(* CODESYS project AnimalCT.project
   Title: AnimalCT
   CompiledLibraryCompatibilityVersion: LeadSysStudio V3.5 SP15 Patch 4

Project tree, tasks and I/O mapping:
  Device : MC508, Leadshine Technology Co., Ltd., order no. 508101, version 3.5.15.40
      settings: RetainMode = 0; RetainStartAddr = 20480; RetainEndAddr = 524288; RetainSize = 524288
    application Application
      libraries: Standard, * (System); CAA SerialCom, 3.5.15.0 (CAA Technical Workgroup); Serial Communication, 3.5.7.0 (3S - Smart Software Solutions GmbH); LS_SysLib, 1.0.0.9 (Leadshine Technology Co.Ltd); CANopenLib, 1.0.0.5 (Leadshine Technology Co.Ltd); CAA Net Base Services, 3.5.15.0 (CAA Technical Workgroup); Network, 3.5.7.0 (3S - Smart Software Solutions GmbH); CANbus, 3.5.7.0 (3S - Smart Software Solutions GmbH); VisuDialogs, * (System); LS_OmronUtils, 1.0.0.2 (Leadshine Technology Co.Ltd); CANopenLib, 1.0.0.5 (Leadshine Technology Co.Ltd); SysMem23, 3.5.13.0 (System); SysFile, 3.5.15.0 (System); SysTypes2 Interfaces, 3.5.4.0 (System)
      task EtherCAT_Master_Leadshine_A (cyclic, interval 4 ms, priority 0) calls EtherCAT_Master_Leadshine_A.EtherCAT_Task, Axis_QJ, Axis_XZ
      task X_Ray (cyclic, interval t#4ms, priority 1) calls DT_Xray
      task MainTask (cyclic, interval 4 ms, priority 1) calls PLC_PRG
      DTU/
        data type E_State
        Axis/
          data type AxisState
          data type AxisCmd
          data type AxisParameter
        TCP/
          data type PLC_SEND
          data type PLC_RECV
          data type Real_TO_Byte_Convert
        data type E_LampCmd
      GVL/
        global variables GVL_Retain
        global variables GVL_SCAN
        global variables GVL_State
      BasicFBs/
        function block Blink [ST]
        function block MoveFilter [ST]
        function block ASCII_Chart_N [ST]
        function block RC [ST]
        function block Curve_Cs [ST]
        function block ASCII_Chart_P [ST]
        function block MeanValue [ST]
        function block Cut [ST]
        function block String2Byte [ST]
      RecordLog/
        program RecordLog [ST]: ACT_RecordState, ACT_RecordError, ACT_RecordCmd, ACT_XrayState, ACT_SysFileOpen, ACT_SysFileRename, ACT_SysFileRead, ACT_SysFileDelete, ACT_SysFileSetPos, ACT_SysFileWrite, ACT_SysFileClose, ACT_SysFileEOF, ACT_SysFileGetPos, ACT_SysFileCopy, ACT_RecordSwitch
      program DT_Xray [SFC]: _Error_active, T_Exp, _Serial_active, T_DR, T_Flu, _aOpenSeria_active, _Exposure1_active, _Wait_active, _Exposure2_entry, _Exposure2_active, _a_Init_active, _QueryState_entry, _Debug_active, _Exposure1_entry, _QueryState_active, _DefaultPara_entry, _DefaultPara_active, _a_DrExposure_active_1, _a_DrExposure_entry_1, _a_DrPara_active_1, _a_DrPara_entry_1, _a_FluoroPara_active_1, _a_FluoroPara_entry_1, _a_FluoroExPosure_active_1, _a_FluoroExPosure_entry_1, _a_ExposurePara_active_1, _a_ExposurePara_entry_1, _a_Exposure_active_1, _a_Exposure_entry_1, _Error_entry, _QueryState_exit, _a_FluoroExPosure_exit
      Refer/
        program Trigger_HaoboPannel [ST]
        program WriteLog [ST]: ACT_SysFileRead, ACT_SysFileDelete, ACT_SysFileClose, ACT_SysFileRename, ACT_SysFileGetPos, ACT_SysFileCopy, ACT_SysFileSetPos, ACT_SysFileEOF, ACT_SysFileWrite, ACT_SysFileOpen
        program XRAY_RS485 [ST]: AXray
      trace Trace (task MainTask): WorkStation_TCP.PLC_RECV1.m_nSocketType, Entity_IO.bXaryOne, Entity_IO.bXaryTwo, Entity_IO.bXaryFlu, Entity_IO.bXrayExp, Entity_IO.bTriggerOut, DT_Xray.RadExp_Step, PLC_PRG.Step_Scout, PLC_PRG.Step_CBCT, WorkStation_TCP.PLC_SEND1.m_nMHuValue, PLC_PRG.Step_StaticDR, WorkStation_TCP.PLC_RECV1.m_nLastMsg, Entity_IO.bXrayOneInput, WorkStation_TCP.PLC_SEND1.m_nMoveState, PLC_PRG.iActNumPulse, PLC_PRG.Step_Air, Entity_IO.bDoorLock, PLC_PRG.Step_QuickCT, GVL_State.iPLC_State
      global variables PersistentVars
      Init/
        program InitMotor [ST]
      visualisation Motor
      program PLC_PRG [SFC]: _a_SelfCheck_active, _a_StandardCT_active, _a_ShutDown_entry_1, T_JUMP_IDLE, _a_StaticDR_exit, _a_Emergercy_active_1, _a_StaticCT_active, _a_Idle_exit, T_StaticDR, T_DynamicsDR, _a_Idle_entry, _a_StaticCT_entry, T_CT, _a_SelfCheck_exit, _a_Error_entry, T_QuickCT, _a_Error_active, _a_HighDefinCT_active, _a_Homing_active, _a_Emergercy_entry_1, _a_QuickCT_exit, T_StandardCT, _a_SelfCheck_entry, AirHigh_entry, T_HighDefinCT, _a_DynamicsDR_exit, _a_Init_active_1, _a_ShutDown_active_1, _a_DynamicsDR_active, _a_Wait_active, _a_Idle_active, _a_Error_exit, _a_HighDefinCT_exit, _a_Homing_entry, _a_Debug_entry, _a_Init_active, _a_Logic_active, _a_Wait_exit, _a_StaticDR_active, _a_QuickCT_entry, _a_StandardCT_entry, _a_StaticCT_exit, _a_SystemInfo_active, _a_HighDefinCT_entry, _a_Debug_active, T_DR, _a_DynamicsDR_entry, _a_Homing_exit, _a_QuickCT_active, _a_MovePos_active, _a_StandardCT_exit, T_StaticCT, _a_StaticDR_entry, AirHigh_active, T_AirCal, T_AirCal_Quick, _AirCalQuick_active, _AirCalQuick_entry, _AirCalHign_exit, _AirCalQuick_exit, _a_Debug_exit, _a_Emergercy_exit, _ModeWait_active
      Logic/
        program WorkMode [ST]
      Motor/
        program Axis_XZ [ST]
        program Axis_QJ [ST]
        program Motor_SJ [ST]
      aSpecailBasic/
        function String2ASCII [ST]
        function block X_RayExpPara [ST]
        function block RecvStringS [ST]
        function block SendStringS [ST]
        function block X_RayFluPara [ST]
        function block String_TO_ASCII [ST]
      visualisation Entity_IO
      Communication/
        program CTBOX_RS232 [ST]
        program Calibration [ST]
        program WorkStation_TCP [ST]: APLC_RECV, APLC_SENG
      IOs/
        program Entity_IO [ST]
    Resource Usage
    Device Diagnose
    Network Configuration
      LocalBus Config
    EtherCAT_Master_Leadshine_A : EtherCAT Master SoftMotion, 3S - Smart Software Solutions GmbH, version 3.5.15.30
        settings: SlaveAutoRestart = True; NetworkName = 'ecat'; SelectNetworkByName = TRUE
      L8EC : L8EC(COE), Leadshine Technology Co.,Ltd., order no. L8EC, version Revision=16#00000001
          settings: StationAlias = 0; DC sync0 cycletime = 4000; DC sync1 cycletime = 4000; Number of SDO = 6; Homing method.Index = 16#6098; Homing method.Subindex = 16#00; Homing method.Value = 13; Homing method.Size = 8; Homing method.AbortIfError = FALSE; Homing method.JumpToLine = FALSE; Homing method.Line = 0; Homing method.CompleteAccess = False; Homing velocity (fast).Index = 16#6099; Homing velocity (fast).Subindex = 16#01; Homing velocity (fast).Value = 82451; Homing velocity (fast).Size = 32; Homing velocity (fast).AbortIfError = FALSE; Homing velocity (fast).JumpToLine = FALSE; Homing velocity (fast).Line = 0; Homing velocity (fast).CompleteAccess = False; Homing velocity (slow).Index = 16#6099; Homing velocity (slow).Subindex = 16#02; Homing velocity (slow).Value = 20612; Homing velocity (slow).Size = 32; Homing velocity (slow).AbortIfError = FALSE; Homing velocity (slow).JumpToLine = FALSE; Homing velocity (slow).Line = 0; Homing velocity (slow).CompleteAccess = False; Homing acceleration.Index = 16#609A; Homing acceleration.Subindex = 16#00; Homing acceleration.Value = 2576613; Homing acceleration.Size = 32; Homing acceleration.AbortIfError = FALSE; Homing acceleration.JumpToLine = FALSE; Homing acceleration.Line = 0; Homing acceleration.CompleteAccess = False; Homing offset.Index = 16#607C; Homing offset.Subindex = 16#00; Homing offset.Value = 0; Homing offset.Size = 32;
            Homing offset.AbortIfError = FALSE; Homing offset.JumpToLine = FALSE; Homing offset.Line = 0; Homing offset.CompleteAccess = False
          input  bRotateMotorMin1 : BOOL  // Digital inputs.Bit0
          input  bRotateMotorMax1 : BOOL  // Digital inputs.Bit1
          unmapped channels: Control word, Profile target position, Touch Probe Function, Servo error code, Last error code, Status word, Modes of operation display, Actual motor position, Touch Probe Status, Touch probe pos1 pos value, Digital inputs
        Axis : Axis, 3S - Smart Software Solutions GmbH, order no. 0, version 4.6.1.0
            settings: wDriveID = 0; dwRatioTechUnitsDenom = 432871; iRatioTechUnitsNum = 42; 一圈脉冲数 = 229167; 工作台一圈的位移 = 360; 电子齿轮比分子 = 340; 电子齿轮比分母 = 21; 回零速度 = 8.000; 回零爬行速度 = 2; 回零加速度 = 250.000; 回零偏移 = 0; 回零速度SDO = 82451; 回零爬行速度SDO = 20612; 回零偏移SDO = 0; ScalingIncs = 229167; ScalingMotorTurns2 = 340; ScalingGearOutput1 = 21; AdrOffset_8010 = 52; BitOffset_8010 = 0; BitLength_8010 = 16; Address_8010 = '%QW26'; Type_8010 = 'UINT'; AddressPointer_8010 = ADR(%QW26); AdrOffset_8020 = 56; BitOffset_8020 = 0; BitLength_8020 = 32; Address_8020 = '%QD14'; Type_8020 = 'DINT'; AddressPointer_8020 = ADR(%QD14); AdrOffset_8030 = 4294967295; BitOffset_8030 = 0; BitLength_8030 = 0; Address_8030 = ''; Type_8030 = ''; AddressPointer_8030 = 0; AdrOffset_8040 = 4294967295; BitOffset_8040 = 0; BitLength_8040 = 0; Address_8040 = ''; Type_8040 = '';
              AddressPointer_8040 = 0; AdrOffset_8050 = 4294967295; BitOffset_8050 = 0; BitLength_8050 = 0; Address_8050 = ''; Type_8050 = ''; AddressPointer_8050 = 0; AdrOffset_8060 = 60; BitOffset_8060 = 0; BitLength_8060 = 16; Address_8060 = '%QW30'; Type_8060 = 'UINT'; AddressPointer_8060 = ADR(%QW30); AdrOffset_8070 = 4294967295; BitOffset_8070 = 0; BitLength_8070 = 0; Address_8070 = ''; Type_8070 = ''; AddressPointer_8070 = 0; AdrOffset_8080 = 4294967295; BitOffset_8080 = 0; BitLength_8080 = 0; Address_8080 = ''; Type_8080 = ''; AddressPointer_8080 = 0; AdrOffset_8090 = 4294967295; BitOffset_8090 = 0; BitLength_8090 = 0; Address_8090 = ''; Type_8090 = ''; AddressPointer_8090 = 0; AdrOffset_8510 = 88; BitOffset_8510 = 0; BitLength_8510 = 16; Address_8510 = '%IW44'; Type_8510 = 'UINT'; AddressPointer_8510 = ADR(%IW44); AdrOffset_8520 = 92; BitOffset_8520 = 0; BitLength_8520 = 32;
              Address_8520 = '%ID23'; Type_8520 = 'DINT'; AddressPointer_8520 = ADR(%ID23); AdrOffset_8530 = 4294967295; BitOffset_8530 = 0; BitLength_8530 = 0; Address_8530 = ''; Type_8530 = ''; AddressPointer_8530 = 0; AdrOffset_8540 = 4294967295; BitOffset_8540 = 0; BitLength_8540 = 0; Address_8540 = ''; Type_8540 = ''; AddressPointer_8540 = 0; AdrOffset_8550 = 90; BitOffset_8550 = 0; BitLength_8550 = 8; Address_8550 = '%IB90'; Type_8550 = 'SINT'; AddressPointer_8550 = ADR(%IB90); AdrOffset_8560 = 104; BitOffset_8560 = 0; BitLength_8560 = 32; Address_8560 = '%ID26'; Type_8560 = 'UDINT'; AddressPointer_8560 = ADR(%ID26); AdrOffset_8570 = 96; BitOffset_8570 = 0; BitLength_8570 = 16; Address_8570 = '%IW48'; Type_8570 = 'UINT'; AddressPointer_8570 = ADR(%IW48); AdrOffset_8580 = 100; BitOffset_8580 = 0; BitLength_8580 = 32; Address_8580 = '%ID25'; Type_8580 = 'DINT'; AddressPointer_8580 = ADR(%ID25); AdrOffset_8590 = 4294967295;
              BitOffset_8590 = 0; BitLength_8590 = 0; Address_8590 = ''; Type_8590 = ''; AddressPointer_8590 = 0; AdrOffset_8600 = 4294967295; BitOffset_8600 = 0; BitLength_8600 = 0; Address_8600 = ''; Type_8600 = ''; AddressPointer_8600 = 0; AdrOffset_8600 = 4294967295; BitOffset_8600 = 0; BitLength_8600 = 0; Address_8610 = ''; Type_8610 = ''; AddressPointer_8610 = 0; AdrOffset_8620 = 4294967295; BitOffset_8620 = 0; BitLength_8620 = 0; Address_8620 = ''; Type_8620 = ''; AddressPointer_8620 = 0; 回零加速度SDO = 2576613
      L8EC_1 : L8EC(COE), Leadshine Technology Co.,Ltd., order no. L8EC, version Revision=16#00000001
          settings: StationAlias = 0; DC sync0 cycletime = 4000; DC sync1 cycletime = 4000; Number of SDO = 6; Homing method.Index = 16#6098; Homing method.Subindex = 16#00; Homing method.Value = 1; Homing method.Size = 8; Homing method.AbortIfError = FALSE; Homing method.JumpToLine = FALSE; Homing method.Line = 0; Homing method.CompleteAccess = False; Homing velocity (fast).Index = 16#6099; Homing velocity (fast).Subindex = 16#01; Homing velocity (fast).Value = 60000; Homing velocity (fast).Size = 32; Homing velocity (fast).AbortIfError = FALSE; Homing velocity (fast).JumpToLine = FALSE; Homing velocity (fast).Line = 0; Homing velocity (fast).CompleteAccess = False; Homing velocity (slow).Index = 16#6099; Homing velocity (slow).Subindex = 16#02; Homing velocity (slow).Value = 12000; Homing velocity (slow).Size = 32; Homing velocity (slow).AbortIfError = FALSE; Homing velocity (slow).JumpToLine = FALSE; Homing velocity (slow).Line = 0; Homing velocity (slow).CompleteAccess = False; Homing acceleration.Index = 16#609A; Homing acceleration.Subindex = 16#00; Homing acceleration.Value = 100000; Homing acceleration.Size = 32; Homing acceleration.AbortIfError = FALSE; Homing acceleration.JumpToLine = FALSE; Homing acceleration.Line = 0; Homing acceleration.CompleteAccess = False
          input  bForeMotorMin1 : BOOL  // Digital inputs.Bit0
          input  bForeMotorMax1 : BOOL  // Digital inputs.Bit1
          unmapped channels: Control word, Profile target position, Touch Probe Function, Servo error code, Last error code, Status word, Modes of operation display, Actual motor position, Touch Probe Status, Touch probe pos1 pos value, Digital inputs
        Axis_1 : Axis, 3S - Smart Software Solutions GmbH, order no. 0, version 4.6.1.0
            settings: dwRatioTechUnitsDenom = 2000; 一圈脉冲数 = 20000; 工作台一圈的位移 = 10; 电子齿轮比分子 = 1; 电子齿轮比分母 = 1; 回零速度 = 30.000; 回零爬行速度 = 6.000; 回零加速度 = 50; 回零偏移 = 0; 回零速度SDO = 60000; 回零爬行速度SDO = 12000; ScalingIncs = 20000; AdrOffset_8010 = 64; BitOffset_8010 = 0; BitLength_8010 = 16; Address_8010 = '%QW32'; Type_8010 = 'UINT'; AddressPointer_8010 = ADR(%QW32); AdrOffset_8020 = 68; BitOffset_8020 = 0; BitLength_8020 = 32; Address_8020 = '%QD17'; Type_8020 = 'DINT'; AddressPointer_8020 = ADR(%QD17); AdrOffset_8030 = 4294967295; BitOffset_8030 = 0; BitLength_8030 = 0; Address_8030 = ''; Type_8030 = ''; AddressPointer_8030 = 0; AdrOffset_8040 = 4294967295; BitOffset_8040 = 0; BitLength_8040 = 0; Address_8040 = ''; Type_8040 = ''; AddressPointer_8040 = 0; AdrOffset_8050 = 4294967295; BitOffset_8050 = 0; BitLength_8050 = 0; Address_8050 = '';
              Type_8050 = ''; AddressPointer_8050 = 0; AdrOffset_8060 = 72; BitOffset_8060 = 0; BitLength_8060 = 16; Address_8060 = '%QW36'; Type_8060 = 'UINT'; AddressPointer_8060 = ADR(%QW36); AdrOffset_8070 = 4294967295; BitOffset_8070 = 0; BitLength_8070 = 0; Address_8070 = ''; Type_8070 = ''; AddressPointer_8070 = 0; AdrOffset_8080 = 4294967295; BitOffset_8080 = 0; BitLength_8080 = 0; Address_8080 = ''; Type_8080 = ''; AddressPointer_8080 = 0; AdrOffset_8090 = 4294967295; BitOffset_8090 = 0; BitLength_8090 = 0; Address_8090 = ''; Type_8090 = ''; AddressPointer_8090 = 0; AdrOffset_8510 = 112; BitOffset_8510 = 0; BitLength_8510 = 16; Address_8510 = '%IW56'; Type_8510 = 'UINT'; AddressPointer_8510 = ADR(%IW56); AdrOffset_8520 = 116; BitOffset_8520 = 0; BitLength_8520 = 32; Address_8520 = '%ID29'; Type_8520 = 'DINT'; AddressPointer_8520 = ADR(%ID29); AdrOffset_8530 = 4294967295; BitOffset_8530 = 0;
              BitLength_8530 = 0; Address_8530 = ''; Type_8530 = ''; AddressPointer_8530 = 0; AdrOffset_8540 = 4294967295; BitOffset_8540 = 0; BitLength_8540 = 0; Address_8540 = ''; Type_8540 = ''; AddressPointer_8540 = 0; AdrOffset_8550 = 114; BitOffset_8550 = 0; BitLength_8550 = 8; Address_8550 = '%IB114'; Type_8550 = 'SINT'; AddressPointer_8550 = ADR(%IB114); AdrOffset_8560 = 128; BitOffset_8560 = 0; BitLength_8560 = 32; Address_8560 = '%ID32'; Type_8560 = 'UDINT'; AddressPointer_8560 = ADR(%ID32); AdrOffset_8570 = 120; BitOffset_8570 = 0; BitLength_8570 = 16; Address_8570 = '%IW60'; Type_8570 = 'UINT'; AddressPointer_8570 = ADR(%IW60); AdrOffset_8580 = 124; BitOffset_8580 = 0; BitLength_8580 = 32; Address_8580 = '%ID31'; Type_8580 = 'DINT'; AddressPointer_8580 = ADR(%ID31); AdrOffset_8590 = 4294967295; BitOffset_8590 = 0; BitLength_8590 = 0; Address_8590 = ''; Type_8590 = ''; AddressPointer_8590 = 0;
              AdrOffset_8600 = 4294967295; BitOffset_8600 = 0; BitLength_8600 = 0; Address_8600 = ''; Type_8600 = ''; AddressPointer_8600 = 0; AdrOffset_8600 = 4294967295; BitOffset_8600 = 0; BitLength_8600 = 0; Address_8610 = ''; Type_8610 = ''; AddressPointer_8610 = 0; AdrOffset_8620 = 4294967295; BitOffset_8620 = 0; BitLength_8620 = 0; Address_8620 = ''; Type_8620 = ''; AddressPointer_8620 = 0; 回零加速度SDO = 100000
    LocalBus_Master_Module : LocalBus Master, Leadshine Technology Co., Ltd., version 3.5.15.40
      PM_3200 : PM_3200, Leadshine Technology Co., Ltd., version 3.5.15.40
          settings: 位置号 = 0
          unmapped channels: ErrorCode, INPUT_0, INPUT_1
      PM0016R : PM0016R, Leadshine Technology Co., Ltd., version 3.5.15.40
          settings: 位置号 = 1
          unmapped channels: ErrorCode, OUTPUT_0
      PM_A0400_IV : PM_A0400_IV, Leadshine Technology Co., Ltd., version 3.5.15.40
          settings: 位置号 = 2; AD0 config.Data_Buffer = 5; AD1 config.Data_Buffer = 5; AD2 config.Data_Buffer = 5; AD3 config.Data_Buffer = 5
          unmapped channels: ErrorCode, ADValue, AnalogDiagnose
    Free_Protocol_RS232_COM : Free Protocol RS232 COM, Leadshine Technology Co., Ltd., version 3.5.15.40
        settings: Vendor.Baudrate = 19200; Vendor.Parity = 2; max send data count = 20; max receive data count = 20; com interval = 25
        unmapped channels: receive control, receive data size, send control, send data size, send data buffer, error status, error id, actual receive data size, actual send data size, receive data
    High_Speed_IO_Module : High Speed IO, Leadshine Technology Co., Ltd., version 3.5.15.40
        settings: HS_IO_Mode_0.High In IO Mode 4 = 196611; HS_IO_Mode_0.High In IO Mode 5 = 196611; Counter_Mask = 48; Ioin_Mask = 1792; HS counter 6.Counter_SetWorkMode = 2; InputFilter Para.Time_In8 = 10; InputFilter Para.Time_In9 = 10; InputFilter Para.Time_In10 = 10
        unmapped channels: Genral_IO_IN, Genral_IO_Out
    SoftMotion General Axis Pool
    Free_Protocol_RS485_COM : Free Protocol RS485 COM, Leadshine Technology Co., Ltd., version 3.5.15.40
        settings: Vendor.Baudrate = 19200; Vendor.Parity = 2; max send data count = 10; max receive data count = 10; com interval = 50
        unmapped channels: receive control, receive data size, send control, send data size, send data buffer, error status, error id, actual receive data size, actual send data size, receive data
  text list GlobalTextList
*)

// Device/Application/DTU/TCP/PLC_SEND
TYPE PLC_SEND:
	STRUCT
		m_nSocketType		:UDINT;	//心跳指令，默认为3，留待判断连接状态。
		m_nCurrentAngle		:REAL;	//为设备当前的旋转角度，单位为角度制下的单位，为度。数精度为1度；
		m_nBedHeight		:REAL;	//为床高，单位为毫米，数据范围为0 - 2000mm；
		m_nBedMovePos		:REAL;	//为床移动距离，以床与探测板的垂直面交线为起点，单位为毫米，数据范围为0 - 3000mm；
		m_nExpStates		:UDINT;	//为曝光状态，枚举值，0:idle（空闲） 1:prep（训机） 2: ready（训机结束，准备完成，可以出束） 3: XrayOn（出射线） 4:XrayOff（关射线） 5 error；
		m_nExpCount			:UDINT;	//为曝光的次数，对应曝光的图像张数；
		m_nFocus			:UDINT;	//按键提示，物理意义更改为按键提示
		m_nMHuValue			:REAL;	//热容量，单位MHu ，实际热容量*100得到，实际热容量为小数；
		m_nDirectionState	:UDINT;	//当前旋转状态，默认值-1， 0为正转，1为反转，停止为-1
		m_nMoveState		:UDINT;	//起始、终止状态， 默认值-1， 0为当前扫描方案（与常规意义不同，注意区别）处于准备好状态，可以准备扫描；1为当前扫描方案结束，运动过程中值为-1
		m_nError			:UDINT;	//错误码使用，由王（风杰）工具体阐述内容
		m_fSpeed			:REAL;	//为设备的旋转速度，单位为度/秒，精度0.01度/秒；
		m_fKv				:UDINT;	//管电压，单位为kv（千伏），精度1；
		m_fMA				:REAL;	//管电流，单位为mA（毫安），精度0.1；
		m_fMs				:REAL;	//曝光时间，单位为ms（毫秒），精度0.01；
		m_nSamplingRate		:UDINT;	//采样率，有3个选项：2400帧/圈；1200帧/圈；600帧/圈
		m_nScanProType		:UDINT;	//执行扫描方案的类型，0为自动扫描，1为手动扫描，2为无设置意义的值，默认值为2
		PLC_State			:UDINT;	//PLC状态
		XRAY_State			:UDINT;	//X射线源状态
		AxisErrorID			:UDINT;	//电机错误标志位，含2个伺服电机
		
		m_nFocusX			:UDINT;	//焦点大小，0为大焦点 1为小焦点， 焦点具体对应的值由plc设置；
		reserve1,reserve2,reserve3,reserve4,reserve5,reserve6,reserve7,reserve8,reserve9:UDINT;
	END_STRUCT
END_TYPE

// Device/Application/DTU/E_State
{attribute 'qualified_only'}
{attribute 'strict'}
TYPE E_State :
(
	初始化		:=10,
	自检		:=20,
	回零		:=30,
	待机 		:=40,
	静态DR		:=110,
	动态DR		:=120,
	标准CT		:=210,
	静态CT 		:=220,
	高清CT		:=230,
	快速CT		:=240,
	错误状态	:=310,
	调试状态 	:=320,
	急停状态	:=330,
	关机状态	:=340
);
END_TYPE

// Device/Application/DTU/TCP/PLC_RECV
TYPE PLC_RECV :
	STRUCT
		m_nSocketType		:UDINT;//0为连接判断信息使用，1为发送设备的有具体意义是参数信息。
      	m_nExpId 			:UDINT;//扫描方式 0为不扫描， 1为静态DR扫描 2为动态DR扫描，3为标准CT，4为静态CT，5为高清CT，6为快速CT
       	m_nAngleStart 		:REAL;//为曝光起始位置，在2D和多次曝光情况下，机架旋转到m_nAngleStart位置后再开始曝光，机架不动；CBCT状态下，机架旋转到m_nAngleStart位置后开始曝光，机架运动至m_nAngleEnd位置；最小值为0。
      	m_nAngleEnd  		:REAL;//为曝光的终止位置，在2D和多次曝光情况下不使用；在CBCT状态下，机架的运动终止位置；最小值为0，最大值为360。
      	m_nRotateBegin  	:REAL;//为旋转的起始位置（考虑加速过程）
      	m_nRotateEnd  		:REAL;//为旋转的终止位置（考虑减速过程）
      	m_nKv  				:UDINT;//设置的管电压值，单位为kv，正整数；
      	m_nMA  				:REAL;//设置的管电流值，单位为mA，正整数；
      	m_nMS 				:REAL;//设置一次曝光的时间，单位为ms（毫秒）；设置一次曝光的时间，单位为us（微秒）；精度为1
       	m_nFocus 			:UDINT;//焦点大小设置，枚举值，0为大焦点， 1小焦点；
      	m_nAcquireFrame 	:UDINT;//总帧数，正整数；
      	m_nFramePerCirCle	:UDINT;//每圈获得的帧数，正整数，帧/圈；
      	m_nMoveToward  		:UDINT;//扫描方向，0为不移动，1为进床方向，2为出床方向；
     	m_nServenLamp  		:UDINT;//七灯是否点亮
      	m_nMoveStep  		:REAL;//步进长度，轴扫时使用，单位为mm（毫米）；
     	m_nPitchValue   	:REAL;//螺距长度，螺旋扫时使用，单位为mm（毫米）；
      	m_nCircleCount  	:UDINT;//旋转总圈数，由起始角度和终止角度计算获得，正整数。
      	m_nControlState 	:UDINT;//控制状态 0为正常 1为中止扫描， 2为退出扫描，默认为0
       	m_fScanTop 			:REAL;//扫描上界，以动物趴卧头朝里的方向为基准，从脚至头方向为正方向。单位为毫米，精度为0.01；
       	m_fScanBottom 		:REAL;//扫描下界，以动物趴卧头朝里的方向为基准，从脚至头方向为正方向。单位为毫米，精度为0.01；
		m_fSecondPerCicle	:REAL;//一圈多少秒
      	m_nSamplingRate  	:UDINT;//采样率，有3个选项：2400帧/圈；1200帧/圈；600帧/圈
       	m_nPrepareState 	:UDINT;//是否亮灯1为亮5灯，0 为不亮5灯
        m_nScanMoveType		:UDINT;//扫描模式 0为手动扫描，1为自动扫描，2为子床位扫描
       	m_nCircleIndex 		:UDINT;//当前第几圈
       	m_nPLCMaCoeff 		:REAL;//灯丝电压值
      	m_nLastMsg  		:UDINT;//CBCT扫描最后一次标志位
       	m_nDelayTime 		:UDINT;//预留
        yuliu_2				:UDINT;//预留
       	yuliu_3 			:UDINT;//预留一共30个数据
	END_STRUCT
END_TYPE

// Device/Application/DTU/E_LampCmd
{attribute 'qualified_only'}
{attribute 'strict'}
TYPE E_LampCmd :
(
	常亮	:=66,
	慢闪	:=22,
	快闪	:=33,
	关闭 	:=55
);
END_TYPE

// Device/Application/DTU/TCP/Real_TO_Byte_Convert
	(*共用体，2个16位WORD和转换为REAL类型*)
	TYPE Real_TO_Byte_Convert :
	UNION
		rData:REAL;					//32字节
		wByte:ARRAY[0..3] OF BYTE;  //8位字节
	END_UNION
	END_TYPE

// Device/Application/DTU/Axis/AxisState
TYPE AxisState :
STRUCT
	bNetState	:BOOL;//网络状态
	bStandStill	:BOOL;//静止状态
	bPowering	:BOOL;//使能状态
	bHoming		:BOOL;//回零状态
	bErrStop	:BOOL;//停止错误
	bStopState	:BOOL;//停止状态
	bAxisErr	:BOOL;//轴故障
	bPowerOff	:BOOL;//轴使能中
	bContinuousMotion:BOOL;//连续运动状态
	bDisCreteMition:BOOL;//离散运动状态
	bSynchronizedMotion:BOOL;//同步运动中
	
	bAxisGoAbsDone	:BOOL;//绝对定位完成10ms后自动复位
	bAxisGoRelDone	:BOOL;//相对定位完成10ms后自动复位
	bResetDone		:BOOL;//复位完成
	
	rActPosition	:LREAL; 	//实际位置
	rActVelocity	:LREAL; 	//实际速度
	rActTorque		:LREAL;	//实际力矩
	rAcc			:REAL;	//加速度数值
	ErrorID			:UDINT;//故障代码
	
END_STRUCT
END_TYPE


(*
	dActPosition	:DINT; 	//实际位置
	dActVelocity	:DINT; 	//实际速度
	dActTorque		:DINT;	//实际力矩
	dAcc			:DINT;	//加速度数值
*)

// Device/Application/DTU/Axis/AxisCmd
TYPE AxisCmd :
STRUCT
	bPower	: BOOL;	//上电使能
	bHome	: BOOL;	//上升沿触发，10ms后自动复位，请勿一致强制ON
	bJogP	: BOOL;	//正向点动
 	bJogN	: BOOL;	//反向点动
	bAbs	: BOOL;	//上升沿触发，10ms后自动复位，请勿一致强制ON
	bRel	: BOOL;	//上升沿触发，10ms后自动复位，请勿一致强制ON
	bVel	: BOOL;  //速度模式 	
	bStop	: BOOL;	//停止
	bReset	: BOOL;//上升沿触发，10ms后自动复位，请勿一致强制ON
	bSetPos	:BOOL;//设置轴当前位置,home
	bSetPosH:BOOL;//setPos
	AxisPara: AxisParameter;
	bSetHomePara:BOOL;//设置回零参数
END_STRUCT
END_TYPE

// Device/Application/DTU/Axis/AxisParameter
TYPE AxisParameter :
STRUCT
	AxisNodeID			: USINT;	
	rZeroOffset			: REAL;//回原点偏移
	rAbsPosition		: REAL;//AxisGoAbs位置
	rAbsVelocity		: REAL;	//AxisGoAbs速度
	rRelVelocity		: REAL;//AxisGoRel速度
	rRelPosition		: REAL;//AxisGoRel位置
	rVelVelocity		: REAL;//AxisVGo速度
	rAccDec				: REAL;//加减速
	rJogVelocity		: REAL;//点动加减速度默认为点动速度10倍
	rSetPosition		: REAL;//设置轴当前位置变量
	
	iHomeMode		:USINT;
	rHomeHighSpeed	:REAL;
	rHomeLowSpeed	:REAL;
	rHomeAcc		:REAL;
END_STRUCT
END_TYPE


(*	
STRUCT
	AxisNodeID			: USINT;	
	dZeroOffset			: UDINT;//回原点偏移
	dAbsPosition		: DINT;//AxisGoAbs位置
	dAbsVelocity		: UDINT;	//AxisGoAbs速度
	dRelVelocity		: UDINT;//AxisGoRel速度
	dRelPosition		: DINT;//AxisGoRel位置
	dVelVelocity		: DINT;//AxisVGo速度
	dAccDec				: UDINT;//加减速
	dJogVelocity		: DINT;//点动加减速度默认为点动速度10倍
	dSetPosition		: UDINT;//设置轴当前位置变量
	
	iHomeMode		:USINT;
	dHomeHighSpeed	:UDINT;
	dHomeLowSpeed	:UDINT;
	dHomeAcc		:UDINT;
END_STRUCT
*)

// Device/Application/GVL/GVL_Retain
{attribute 'qualified_only'}

VAR_GLOBAL PERSISTENT RETAIN
	rBedRecordHeight:REAL;//断电保存
	rBedRecordLength:REAL;//断电保存
	
	rXZ_Zero:REAL;
	rSJ_Zero:INT;
	
	
	rXZ_Position:REAL;
	rQJ_Position:REAL;
END_VAR

// Device/Application/GVL/GVL_SCAN
{attribute 'qualified_only'}
VAR_GLOBAL
		bJumpScan:BOOL;
END_VAR

// Device/Application/PersistentVars
{attribute 'qualified_only'}	//掉电保持数据

// Device/Application/GVL/GVL_State
{attribute 'qualified_only'}
VAR_GLOBAL
		iPLC_State:UDINT;
		
		iXray_State:UDINT; 
	
END_VAR

// Device/Application/Motor/Axis_QJ
PROGRAM Axis_QJ
VAR
	
	fbMC_Power			:	MC_Power;
	fbMC_Jog			: 	MC_Jog;
	fbMC_Stop			: 	MC_STOP;	
	fbMC_Home			:	MC_HOME;
	fbMC_Reset			:	MC_Reset;
	fbMC_MoveAbsolute	: 	MC_MoveAbsolute;
	fbMC_MoveRelative	: 	MC_MoveRelative;
	fbMC_ReadStatus		:	MC_ReadStatus;
	fbMC_ReadActualPosition:MC_ReadActualPosition;
	fbMC_ReadActualVelocity	:MC_ReadActualVelocity;
	fbMC_ReadActualTorque:MC_ReadActualTorque;
	fbMC_MoveVelocity:MC_MoveVelocity;
	fbMC_SetPostiong:		MC_SetPosition;
	count				:	BYTE;
	VelDirection:INT:=1;
END_VAR

VAR_INPUT
	QJ_AxisCmd			:AxisCmd;
END_VAR

VAR_OUTPUT	
	QJ_AxisState 		:AxisState;
END_VAR

(*--------------README----------*)
(*旋转电机运动子程序*)

(*1.心跳*)
	count:=count+1;
				
(*2.判断电机轴状态*)
	fbMC_ReadStatus(Axis:= AXIS_1, Enable:= TRUE , //周期刷新
					valid=> , 
					Busy=> , 
					Error=> QJ_AxisState.bAxisErr,   	//轴错误
					ErrorID=> QJ_AxisState.ErrorID,  	//错误ID
					ErrorStop=>QJ_AxisState.bErrStop , 	//轴停止
					Disabled=> QJ_AxisState.bPowerOff, 	//轴未使能
					stopping=> QJ_AxisState.bStopState, //轴紧急停止
					Homing=>	QJ_AxisState.bHoming , 		//回零中
					Standstill=> QJ_AxisState.bStandStill, //使能中
					DiscreteMotion=> QJ_AxisState.bDisCreteMition, 		//离散运动中
					ContinuousMotion=>QJ_AxisState.bContinuousMotion );	//持续运动中
					
		
(*3 读取轴当前位置、速度*)
(*3.1 获取当前位置*)
	fbMC_ReadActualPosition(
								Axis:= AXIS_1, 
								Enable:= TRUE, 
								Valid=> , 
								Busy=> , 
								Error=> , 
								ErrorID=> , 
								Position=> QJ_AxisState.rActPosition);
(*3.2 获取当前速度*)	
	fbMC_ReadActualVelocity(
								Axis:= AXIS_1 ,
								Enable:= TRUE, 
								Valid=> , 
								Busy=> , 
								Error=> , 
								ErrorID=> , 
								Velocity=> QJ_AxisState.rActVelocity);
(*3.3 获取当前力矩*)								
	fbMC_ReadActualTorque(
								Axis:= AXIS_1 ,
								Enable:= TRUE, 
								Valid=> , 
								Busy=> , 
								Error=> , 
								ErrorID=> , 
								Torque=> );
	QJ_AxisState.rActTorque:=fbMC_ReadActualTorque.Torque*1270/1000;						
(*4.使能*)
	fbMC_Power(
				Axis:= AXIS_1 ,
				Enable:= TRUE, 
				bRegulatorOn:= QJ_AxisCmd.bPower,  
				bDriveStart:= QJ_AxisCmd.bPower,  
				Status=>  QJ_AxisState.bPowering, 
				bRegulatorRealState=> , 
				bDriveStartRealState=> , 
				Busy=> , 
				Error=> , 
				ErrorID=> );
	
(*5.回零*)
	fbMC_Home(
				Axis:= AXIS_1, 
				Execute:= QJ_AxisCmd.bHome, 
				Position:= 0,				//回零模式1，默认写零
				Done=> , 
				Busy=> , 
				CommandAborted=> , 
				Error=> , 
				ErrorID=> );
				
(*6.设置当前位置*)			
	fbMC_SetPostiong(
						Axis:= AXIS_1, 
						Execute:= QJ_AxisCmd.bSetPos, 
						Position:= GVL_Retain.rQJ_Position, //设置当前位置
						Mode:= FALSE, 
						Done=> , 
						Busy=> , 
						Error=> , 
						ErrorID=> );
	
(*6.速度模式*)
(*	IF QJ_AxisCmd.AxisPara.rVelVelocity>0 THEN
			VelDirection:=1;
		ELSE
			VelDirection:=-1;
		END_IF
	fbMC_MoveVelocity(
					Axis:=AXIS_1 , 
					Execute:=  QJ_AxisCmd.bVel, 
					Velocity:=ABS(QJ_AxisCmd.AxisPara.rVelVelocity), 
					Acceleration:= QJ_AxisCmd.AxisPara.rAccDec, 
					Deceleration:= QJ_AxisCmd.AxisPara.rAccDec, 
					Jerk:= QJ_AxisCmd.AxisPara.rAccDec*10, 
					Direction:= VelDirection, 
					BufferMode:= 0, 
					InVelocity=> , 
					Busy=> , 
					Active=> , 
					CommandAborted=> , 
					Error=> , 
					ErrorID=> );
*)
(*7.轴绝对运动*)
	fbMC_MoveAbsolute(
						Axis:= AXIS_1, 
						Execute:= QJ_AxisCmd.bAbs AND (NOT QJ_AxisState.bStopState), 
						Position:= QJ_AxisCmd.AxisPara.rAbsPosition, 
						Velocity:= QJ_AxisCmd.AxisPara.rAbsVelocity, 
						Acceleration:= QJ_AxisCmd.AxisPara.rAccDec, 
						Deceleration:= QJ_AxisCmd.AxisPara.rAccDec, 
						Jerk:= QJ_AxisCmd.AxisPara.rAccDec*10, 
						Direction:= 1, 
						BufferMode:= 0, 
						Done=> , 
						Busy=> , 
						Active=> , 
						CommandAborted=> , 
						Error=> , 
						ErrorID=> );
	
						
(*8.轴相对运动*)
	fbMC_MoveRelative(
						Axis:= AXIS_1, 
						Execute:= QJ_AxisCmd.bRel, 
						Distance:= QJ_AxisCmd.AxisPara.rRelPosition, 
						Velocity:=  QJ_AxisCmd.AxisPara.rRelVelocity, 
						Acceleration:=  QJ_AxisCmd.AxisPara.rAccDec, 
						Deceleration:=  QJ_AxisCmd.AxisPara.rAccDec, 
						Jerk:= QJ_AxisCmd.AxisPara.rAccDec*10, 
						BufferMode:= 0, //中断
						Done=> , 
						Busy=> , 
						Active=> , 
						CommandAborted=> , 
						Error=> , 
						ErrorID=> );
						
(*9.轴点动*)
	fbMC_Jog(
				Axis:= AXIS_1 ,
				JogForward:=  QJ_AxisCmd.bJogP AND (NOT QJ_AxisCmd.bJogN),
				JogBackward:= QJ_AxisCmd.bJogN AND (NOT QJ_AxisCmd.bJogP),
				Velocity:= QJ_AxisCmd.AxisPara.rJogVelocity,
				Acceleration:= QJ_AxisCmd.AxisPara.rAccDec, 
				Deceleration:= QJ_AxisCmd.AxisPara.rAccDec, 
				Jerk:= QJ_AxisCmd.AxisPara.rAccDec*10, 
				Busy=> , 
				CommandAborted=> , 
				Error=> , 
				ErrorId=> );

(*10.轴停止*)
	fbMC_Stop(
				Axis:= AXIS_1 ,
				Execute:=  QJ_AxisCmd.bStop, 
				Deceleration:= QJ_AxisCmd.AxisPara.rAccDec, 
				Jerk:= QJ_AxisCmd.AxisPara.rAccDec*10, 
				Done=> , 
				Busy=> , 
				Error=> , 
				ErrorID=> );

	IF fbMC_Stop.Done OR fbMC_Stop.Error THEN
		QJ_AxisCmd.bStop:=FALSE;
	END_IF

(*11.轴复位*)
	fbMC_Reset(
				Axis:= AXIS_1, 
				Execute:= QJ_AxisCmd.bReset, 
				Done=> QJ_AxisState.bResetDone, 
				Busy=> , 
				Error=> , 
				ErrorID=> );

END_PROGRAM

// Device/Application/Motor/Axis_XZ
PROGRAM Axis_XZ
VAR
	
	fbMC_Power			:	MC_Power;
	fbMC_Jog			: 	MC_Jog;
	fbMC_Stop			: 	MC_STOP;	
	fbMC_Home			:	MC_HOME;
	fbMC_Reset			:	MC_Reset;
	fbMC_MoveAbsolute	: 	MC_MoveAbsolute;
	fbMC_MoveRelative	: 	MC_MoveRelative;
	fbMC_ReadStatus		:	MC_ReadStatus;
	fbMC_ReadActualPosition:MC_ReadActualPosition;
	fbMC_ReadActualVelocity	:MC_ReadActualVelocity;
	fbMC_ReadActualTorque	:MC_ReadActualTorque;
	fbMC_MoveVelocity:		MC_MoveVelocity;
	fbMC_SetPostiong:		MC_SetPosition;
	VelDirection:INT:=1;
	count				:	BYTE;
	rLoadTorque:REAL;//负载力矩
END_VAR

VAR_INPUT
	XZ_AxisCmd			:AxisCmd;
END_VAR

VAR_OUTPUT	
	XZ_AxisState 		:AxisState;
END_VAR

(*--------------README----------*)
(*旋转电机运动子程序*)

(*1.心跳*)
	count:=count+1;
				
(*2.判断电机轴状态*)
	fbMC_ReadStatus(Axis:= Axis, Enable:= TRUE , //周期刷新
					valid=> , 
					Busy=> , 
					Error=> XZ_AxisState.bAxisErr,   	//轴错误
					ErrorID=> XZ_AxisState.ErrorID,  	//错误ID
					ErrorStop=>XZ_AxisState.bErrStop , 	//轴停止
					Disabled=> XZ_AxisState.bPowerOff, 	//轴未使能
					stopping=> XZ_AxisState.bStopState, //轴紧急停止
					Homing=>XZ_AxisState.bHoming , 		//回零中
					Standstill=> XZ_AxisState.bStandStill, //使能中
					DiscreteMotion=> XZ_AxisState.bDisCreteMition, 		//离散运动中
					ContinuousMotion=>XZ_AxisState.bContinuousMotion );	//持续运动中
					
		
(*3 读取轴当前位置、速度*)
(*3.1 获取当前位置*)
	fbMC_ReadActualPosition(
								Axis:= AXIS, 
								Enable:= TRUE, 
								Valid=> , 
								Busy=> , 
								Error=> , 
								ErrorID=> , 
								Position=> XZ_AxisState.rActPosition);
(*3.2 获取当前速度*)	
	fbMC_ReadActualVelocity(
								Axis:= AXIS, 
								Enable:= TRUE, 
								Valid=> , 
								Busy=> , 
								Error=> , 
								ErrorID=> , 
								Velocity=> XZ_AxisState.rActVelocity);
(*3.3 获取当前力矩*)								
	fbMC_ReadActualTorque(
								Axis:= AXIS, 
								Enable:= TRUE, 
								Valid=> , 
								Busy=> , 
								Error=> , 
								ErrorID=> , 
								Torque=> );
	XZ_AxisState.rActTorque:=fbMC_ReadActualTorque.Torque*2390/1000;//换算成mNM,额定力矩2.39NM ,反馈0.1%
	
	rLoadTorque:=LREAL_TO_REAL(XZ_AxisState.rActTorque)*371/1000;
								
(*4.使能*)
	fbMC_Power(
				Axis:= AXIS, 
				Enable:= TRUE, 
				bRegulatorOn:=  XZ_AxisCmd.bPower, 
				bDriveStart:=  XZ_AxisCmd.bPower, 
				Status=> XZ_AxisState.bPowering, 
				bRegulatorRealState=> , 
				bDriveStartRealState=> , 
				Busy=> , 
				Error=> , 
				ErrorID=> );
	
(*5.回零*)
	fbMC_Home(
				Axis:= AXIS, 
				Execute:= XZ_AxisCmd.bHome, 
				Position:= GVL_Retain.rXZ_Zero, 
				Done=> , 
				Busy=> , 
				CommandAborted=> , 
				Error=> , 
				ErrorID=> );
	
(*6.设置当前位置*)
	fbMC_SetPostiong(
						Axis:= AXIS, 
						Execute:= XZ_AxisCmd.bSetPos, 
						Position:= GVL_Retain.rXZ_Position, 
						Mode:= FALSE, 
						Done=> , 
						Busy=> , 
						Error=> , 
						ErrorID=> );
(*6.速度模式*)
(*	IF XZ_AxisCmd.AxisPara.rVelVelocity>0 THEN
		VelDirection:=1;
	ELSE
		VelDirection:=-1;
	END_IF
	fbMC_MoveVelocity(
				Axis:=AXIS , 
				Execute:=  XZ_AxisCmd.bVel, 
				Velocity:= ABS(XZ_AxisCmd.AxisPara.rVelVelocity), 
				Acceleration:= XZ_AxisCmd.AxisPara.rAccDec, 
				Deceleration:= XZ_AxisCmd.AxisPara.rAccDec, 
				Jerk:= XZ_AxisCmd.AxisPara.rAccDec*10, 
				Direction:= VelDirection, 
				BufferMode:= 0, 
				InVelocity=> , 
				Busy=> , 
				Active=> , 
				CommandAborted=> , 
				Error=> , 
				ErrorID=> );
*)
(*7.轴绝对运动*)
	fbMC_MoveAbsolute(
						Axis:= Axis, 
						Execute:= XZ_AxisCmd.bAbs AND (NOT XZ_AxisState.bStopState), 
						Position:= XZ_AxisCmd.AxisPara.rAbsPosition, 
						Velocity:= XZ_AxisCmd.AxisPara.rAbsVelocity, 
						Acceleration:= XZ_AxisCmd.AxisPara.rAccDec, 
						Deceleration:= XZ_AxisCmd.AxisPara.rAccDec, 
						Jerk:= XZ_AxisCmd.AxisPara.rAccDec*10, 
						Direction:= 1, 
						BufferMode:= 0, 
						Done=> , 
						Busy=> , 
						Active=> , 
						CommandAborted=> , 
						Error=> , 
						ErrorID=> );
	
						
(*8.轴相对运动*)
	fbMC_MoveRelative(
						Axis:= Axis, 
						Execute:= XZ_AxisCmd.bRel, 
						Distance:= XZ_AxisCmd.AxisPara.rRelPosition, 
						Velocity:=  XZ_AxisCmd.AxisPara.rRelVelocity, 
						Acceleration:=  XZ_AxisCmd.AxisPara.rAccDec, 
						Deceleration:=  XZ_AxisCmd.AxisPara.rAccDec, 
						Jerk:= XZ_AxisCmd.AxisPara.rAccDec*10, 
						BufferMode:= 0, //中断
						Done=> , 
						Busy=> , 
						Active=> , 
						CommandAborted=> , 
						Error=> , 
						ErrorID=> );
						
(*9.轴点动*)
	fbMC_Jog(
				Axis:= AXIS, 
				JogForward:=  XZ_AxisCmd.bJogP AND (NOT XZ_AxisCmd.bJogN),
				JogBackward:= XZ_AxisCmd.bJogN AND (NOT XZ_AxisCmd.bJogP),
				Velocity:= XZ_AxisCmd.AxisPara.rJogVelocity,
				Acceleration:= XZ_AxisCmd.AxisPara.rAccDec, 
				Deceleration:= XZ_AxisCmd.AxisPara.rAccDec, 
				Jerk:= XZ_AxisCmd.AxisPara.rAccDec*10, 
				Busy=> , 
				CommandAborted=> , 
				Error=> , 
				ErrorId=> );

(*10.轴停止*)
	fbMC_Stop(
				Axis:= AXIS, 
				Execute:=  XZ_AxisCmd.bStop, 
				Deceleration:= XZ_AxisCmd.AxisPara.rAccDec, 
				Jerk:= XZ_AxisCmd.AxisPara.rAccDec*10, 
				Done=> , 
				Busy=> , 
				Error=> , 
				ErrorID=> );

	IF fbMC_Stop.Done OR fbMC_Stop.Error THEN
		XZ_AxisCmd.bStop:=FALSE;
	END_IF

(*11.轴复位*)
	fbMC_Reset(
				Axis:= Axis, 
				Execute:= XZ_AxisCmd.bReset, 
				Done=> XZ_AxisState.bResetDone, 
				Busy=> , 
				Error=> , 
				ErrorID=> );

END_PROGRAM

// Device/Application/DT_Xray
PROGRAM DT_Xray
VAR
	Open_0: COM.Open;
	Write_0: COM.Write;
	Read_0: COM.Read;
	Close_0: COM.Close;
	hComHandle:CAA.HANDLE;
	aParamsB19200 : ARRAY [1..7] OF COM.PARAMETER := [
    (udiParameterId := COM.CAA_Parameter_Constants.udiPort,udiValue := 3), 					//指令端口2,3,4,5分别对应硬件接口com2、com0、com1、com3
    (udiParameterId := COM.CAA_Parameter_Constants.udiBaudrate,udiValue := 19200),			//波特率，设置为19200
    (udiParameterId := COM.CAA_Parameter_Constants.udiParity,udiValue := COM.PARITY.NONE),	//校验，设置为无校验
    (udiParameterId := COM.CAA_Parameter_Constants.udiStopBits,udiValue := COM.STOPBIT.ONESTOPBIT),//停止位，1位
    (udiParameterId := COM.CAA_Parameter_Constants.udiTimeout,udiValue := 500),				//超时时间，设置成500ms
    (udiParameterId := COM.CAA_Parameter_Constants.udiByteSize,udiValue := 8),				//数据位
    (udiParameterId := COM.CAA_Parameter_Constants.udiBinary, udiValue := 1)				//二进制参数，启用二进制模式
];		
	bSend: BOOL;//发送触发
	TON1,TON2,TON3:Standard.TON;//延迟打开串口，读取状态周期，初始态故障复位
	byReadData:ARRAY [0..255] OF BYTE; //读取串口数据
	xClose_Exe: BOOL; //关闭串口操作
	
	ReadString:RecvStringS;//读取射线源反馈，并转化为字符串型数据
	
	Lookup_Step:INT:=0;//查询状态的轮询
	BLINK1,BLINK1_ST,BLINK1_1S:Blink;
	
	SendStringS1:SendStringS;//单命令字符串发送
	
	ASCII_Chart_N2:ARRAY[0..30] OF ASCII_Chart_N;//解析查询态下的ASCII
	ASCII_Chart_N_Alarm:ARRAY[0..5] OF ASCII_Chart_N;//解析报警状态下的故障码
	ASCII_Chart_N_Alarm1,ASCII_Chart_N_Alarm2,ASCII_Chart_N_Alarm3:ASCII_Chart_N;
	(*透视写参变量*)
	FluParaSet:X_RayFluPara;//透视模式下的大指令写入
	String_TO_ASCII1:String_TO_ASCII;	//大命令字符串转化为ASCII码，给计算和校验用的
	ArrASCII:ARRAY[1..255] OF BYTE;		//ASCII放到数组里	
	CheckSum,CheckSum1,CheckSum2:UINT;//和校验处理
	CheckSum3,CheckSum4,CheckSum5:UINT;//和校验处理
	CheckSumString:STRING;//计算后的和校验后1个byte转化为字符串类型
	j,k:INT;//计算和校验用的//HE热量
	sSendStringFlu:STRING;//发送透视模式下的大命令
	TON_HangOver:TON;
	
	(*曝光写参变量*)
	ExpParaSet:X_RayExpPara;//透视模式下的大指令写入
	R_TRIG1,R_TRIG2,R_TRIG3,R_TRIG4,R_TRIG5,R1,R2,R3,R_Error:R_TRIG;
	bXrayError,bXrayError1: BOOL;//射线源出错标志位
	iDR_Staiton:UINT; //DR模式下的BU0选择，选择不同的站模式
	TON11,TON12,TON13,TON14:TON;//曝光跳出
	TOF11:TOF;
	bJumpRadExp:BOOL;
	
	Step_Error:INT;//错误回复步骤
	TOF_DR1:Standard.TOF;//延迟断电继电器控制
	
	
	bResetXray1:BOOL;
	bResetXray2:BOOL;
	sResetError,sResetError1,sResetError2,sResetError3,sResetError4:STRING;
END_VAR

VAR_OUTPUT
	iXray_State:INT;//射线源状态，改用全局变量
	Init_Step,Default_Step,Query_Step,RadExp_Step,RadFlu_Step,ExpPara_Step,FluPara_Setp,DR_Step,DR_Para:INT;//子状态
	Feedback_Kv:UDINT;
	Feedback_mA:REAL;
	Feedback_ms:REAL;
	Feedback_nFocus:UDINT;
	Feedback_nMHuValue:REAL;
	Feedback_AccTime:REAL;
	iAlarmNum:UINT;		//射线源部分的报警位
END_VAR

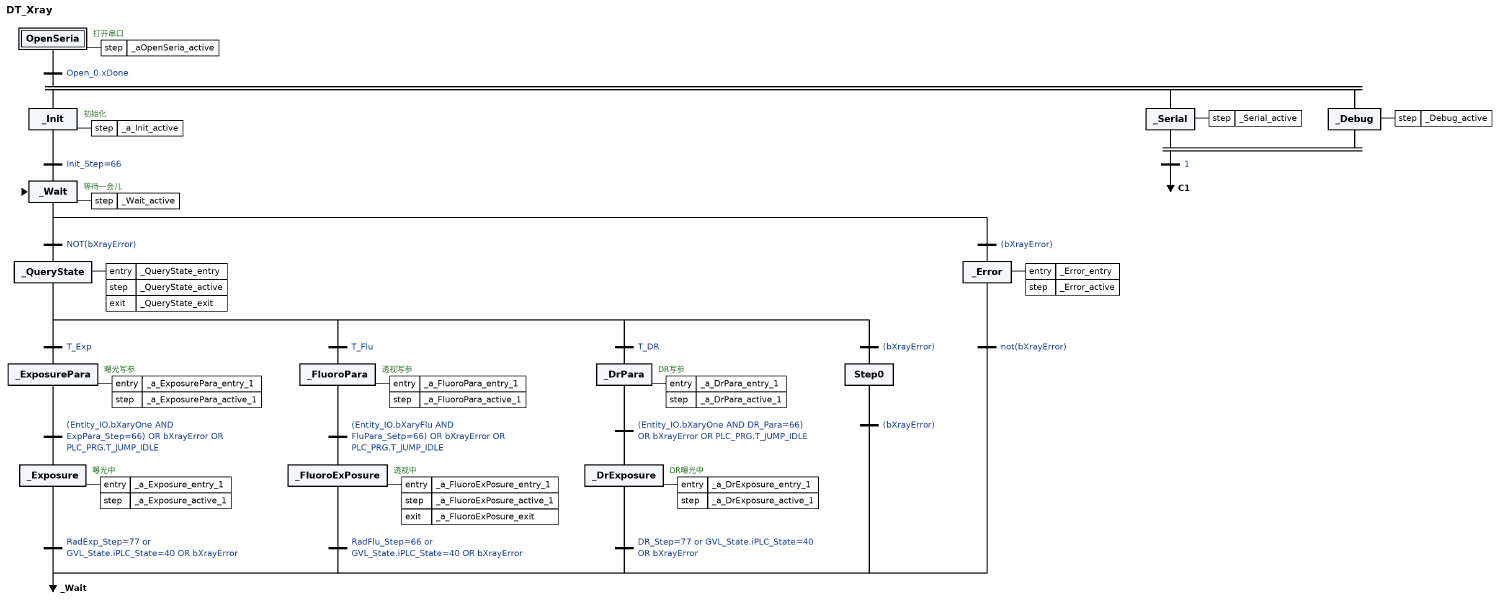
// 打开串口
INITIAL_STEP OpenSeria:
    _aOpenSeria_active(N);  // step action
END_STEP
TRANSITION FROM OpenSeria TO (_Init, _Serial, _Debug)
    := Open_0.xDone;
END_TRANSITION
// 初始化
STEP _Init:
    _a_Init_active(N);  // step action
END_STEP
TRANSITION FROM _Init TO _Wait
    := Init_Step=66;
END_TRANSITION
// 等待一会儿
STEP _Wait:
    _Wait_active(N);  // step action
END_STEP
TRANSITION FROM _Wait TO _QueryState
    := NOT(bXrayError);
END_TRANSITION
STEP _QueryState:
    _QueryState_entry(P1);  // entry action
    _QueryState_active(N);  // step action
    _QueryState_exit(P0);  // exit action
END_STEP
TRANSITION FROM _QueryState TO _ExposurePara
    := T_Exp;
END_TRANSITION
// 曝光写参
STEP _ExposurePara:
    _a_ExposurePara_entry_1(P1);  // entry action
    _a_ExposurePara_active_1(N);  // step action
END_STEP
TRANSITION FROM _ExposurePara TO _Exposure
    := (Entity_IO.bXaryOne AND ExpPara_Step=66) OR bXrayError OR PLC_PRG.T_JUMP_IDLE;
END_TRANSITION
// 曝光中
STEP _Exposure:
    _a_Exposure_entry_1(P1);  // entry action
    _a_Exposure_active_1(N);  // step action
END_STEP
TRANSITION FROM _Exposure TO _Wait
    := RadExp_Step=77 or GVL_State.iPLC_State=40 OR bXrayError;
END_TRANSITION
TRANSITION FROM _QueryState TO _FluoroPara
    := T_Flu;
END_TRANSITION
// 透视写参
STEP _FluoroPara:
    _a_FluoroPara_entry_1(P1);  // entry action
    _a_FluoroPara_active_1(N);  // step action
END_STEP
TRANSITION FROM _FluoroPara TO _FluoroExPosure
    := (Entity_IO.bXaryFlu AND FluPara_Setp=66) OR bXrayError OR PLC_PRG.T_JUMP_IDLE;
END_TRANSITION
// 透视中
STEP _FluoroExPosure:
    _a_FluoroExPosure_entry_1(P1);  // entry action
    _a_FluoroExPosure_active_1(N);  // step action
    _a_FluoroExPosure_exit(P0);  // exit action
END_STEP
TRANSITION FROM _FluoroExPosure TO _Wait
    := RadFlu_Step=66 or GVL_State.iPLC_State=40 OR bXrayError;
END_TRANSITION
TRANSITION FROM _QueryState TO _DrPara
    := T_DR;
END_TRANSITION
// DR写参
STEP _DrPara:
    _a_DrPara_entry_1(P1);  // entry action
    _a_DrPara_active_1(N);  // step action
END_STEP
TRANSITION FROM _DrPara TO _DrExposure
    := (Entity_IO.bXaryOne AND DR_Para=66) OR bXrayError OR PLC_PRG.T_JUMP_IDLE;
END_TRANSITION
// DR曝光中
STEP _DrExposure:
    _a_DrExposure_entry_1(P1);  // entry action
    _a_DrExposure_active_1(N);  // step action
END_STEP
TRANSITION FROM _DrExposure TO _Wait
    := DR_Step=77 or GVL_State.iPLC_State=40 OR bXrayError;
END_TRANSITION
TRANSITION FROM _QueryState TO Step0
    := (bXrayError);
END_TRANSITION
STEP Step0:
END_STEP
TRANSITION FROM Step0 TO _Wait
    := (bXrayError);
END_TRANSITION
TRANSITION FROM _Wait TO _Error
    := (bXrayError);
END_TRANSITION
STEP _Error:
    _Error_entry(P1);  // entry action
    _Error_active(N);  // step action
END_STEP
TRANSITION FROM _Error TO _Wait
    := not(bXrayError);
END_TRANSITION
STEP _Serial:
    _Serial_active(N);  // step action
END_STEP
STEP _Debug:
    _Debug_active(N);  // step action
END_STEP
TRANSITION FROM (_Serial, _Debug) TO (_Serial, _Debug)
    := 1;
END_TRANSITION
// branch label C1
// branch label B1

ACTION _Error_active:
	
	(*EL036故障清除，曝光模式下定位像，没有收到PR1,此时报EL036，需要再发PR0才能彻底清除*)
(*	
	IF (byReadData[0]=16#45 AND byReadData[1]=16#4C)	THEN
		CASE Step_Error OF
			0:	
				R1(CLK:=FALSE , Q=> );	R2(CLK:=FALSE , Q=> );	R3(CLK:=FALSE , Q=> );
				Step_Error:=10;
			10:
				SendStringS1.sSendStringS:=ReadString.RecvString;
				R1(CLK:=(byReadData[0]=16#45 AND byReadData[1]=16#4C) , Q=>bSend );
				IF bSend THEN
					Step_Error:=20;
				END_IF
			20:
				SendStringS1.sSendStringS:='PR0';
				//R2(CLK:=(byReadData[0]=16#45 AND byReadData[1]=16#4C) , Q=>bSend );
				Step_Error:=0;
		END_CASE
	ELSE
		Step_Error:=0;
	END_IF
*)
END_ACTION

TRANSITION T_Exp:


		 
(*下发了指令，并且不是强制退出指令*)
(*DR模式走曝光状态*)		 
(WorkStation_TCP.PLC_RECV1.m_nSocketType=1 AND WorkStation_TCP.PLC_RECV1.m_nControlState=0) 
AND ( WorkStation_TCP.PLC_RECV1.m_nExpId=4 OR WorkStation_TCP.PLC_RECV1.m_nExpId=6 OR WorkStation_TCP.PLC_RECV1.m_nExpId=8)
AND  GVL_State.iPLC_State<>40


(*WorkStation_TCP.PLC_RECV1.m_nExpId=3*)
END_TRANSITION

ACTION _Serial_active:
(*-------------------------------串口基本操作-------------------------------*)

(*1.Write*)
	Write_0(
			xExecute:= Open_0.xDone AND bSend, 
			xAbort:= , 
			udiTimeOut:=500 , 
			xDone=> , 
			xBusy=> , 
			xError=> , 
			xAborted=> , 
			hCom:= hComHandle, 
			pBuffer:= , //后面写的
			szSize:= , 
			eError=> );	
			
(*2.Read*)
	TON2(IN:=NOT TON2.Q , PT:=T#20MS , Q=> , ET=> );	//射线源周期100ms
	Read_0(
			xExecute:= Open_0.xDone AND TON2.Q AND NOT(bSend),
			xAbort:= , 
			udiTimeOut:= 500, 
			xDone=> , 
			xBusy=> , 
			xError=> , 
			xAborted=> , 
			hCom:= hComHandle,
			pBuffer:= ADR(byReadData), 
			szBuffer:= 30, 
			eError=> , 
			szSize=> );
	
(*3.Close*)
	Close_0(
			xExecute:= xClose_Exe, 
			xDone=> , 
			xBusy=> , 
			xError=> , 
			hCom:= hComHandle, 
			eError=> );
			
(*4.读取*)			
	ReadString(Excute:= Read_0.xDone AND Read_0.szSize<>0, Size:=__UXINT_TO_INT(Read_0.szSize) , RecvArray:=byReadData , RecvString=> );

(*5.*)	
	BLINK1_ST(ENABLE:=TON1.Q , TIMELOW:=T#2S , TIMEHIGH:=T#2S , OUT=> );
	BLINK1(ENABLE:=TON1.Q , TIMELOW:=T#200MS , TIMEHIGH:=T#200MS , OUT=> );
	BLINK1_1S(ENABLE:=TON1.Q , TIMELOW:=T#1S , TIMEHIGH:=T#1S , OUT=> );
END_ACTION

TRANSITION T_DR:


(WorkStation_TCP.PLC_RECV1.m_nSocketType=1 AND WorkStation_TCP.PLC_RECV1.m_nControlState=0) AND (WorkStation_TCP.PLC_RECV1.m_nExpId=1 OR WorkStation_TCP.PLC_RECV1.m_nExpId=2 )
END_TRANSITION

TRANSITION T_Flu:


(*下发了指令，并且不是强制退出指令*)		 
(WorkStation_TCP.PLC_RECV1.m_nSocketType=1 AND WorkStation_TCP.PLC_RECV1.m_nControlState=0) AND (WorkStation_TCP.PLC_RECV1.m_nExpId=3 OR WorkStation_TCP.PLC_RECV1.m_nExpId=5 OR WorkStation_TCP.PLC_RECV1.m_nExpId=7)
AND  GVL_State.iPLC_State<>40
END_TRANSITION

ACTION _aOpenSeria_active:



(*1.open*)
	TON1(IN:=TRUE , PT:=T#5S);//开机后5秒打开串口
	Open_0(xExecute:=TON1.Q , xDone=> , xBusy=> , xError=> , usiListLength:=20 , pParameterList:=ADR(aParamsB19200) , eError=> , hCom=>hComHandle );//20??

(*射线源状态*)
	GVL_State.iXray_State:=10;
END_ACTION

ACTION _Exposure1_active:


IF Entity_IO.bXaryOne=FALSE AND Entity_IO.bXaryTwo=FALSE THEN
	IF ReadString.RecvString='PR0' THEN // PR0
		SendStringS1.sSendStringS:='PR0';//曝光完成
		R_TRIG3(CLK:= ReadString.RecvString='PR0', Q=>bSend );//收到立刻发送
		bJumpRadExp:=TRUE;
	END_IF; 
END_IF
END_ACTION

ACTION _Wait_active:
;
END_ACTION

ACTION _Exposure2_entry:
RadExp_Step:=0;
END_ACTION

ACTION _Exposure2_active:
	



	CASE RadExp_Step OF
		0:
			bSend:=FALSE;R_TRIG1(CLK:=FALSE);R_TRIG2(CLK:=FALSE);R_TRIG3(CLK:=FALSE);R_TRIG4(CLK:=FALSE);
			TON13(IN:=FALSE);
			RadExp_Step:=5;

		5:	//
			IF ReadString.RecvString='PR0' THEN // PR1
				SendStringS1.sSendStringS:='PR0';//一档信号
				R_TRIG1(CLK:=ReadString.RecvString='PR0' , Q=>bSend );//收到立刻发送	
			END_IF;
			
			IF ReadString.RecvString='PR0' THEN
				RadExp_Step:=10;
			END_IF;
			
		10:
			IF ReadString.RecvString='PR0' THEN // PR2
				SendStringS1.sSendStringS:='PR0';//阳极加速完成 
				R_TRIG2(CLK:=ReadString.RecvString='PR0' , Q=>bSend );//收到立刻发送
			END_IF;
			
			IF ReadString.RecvString='PR0' THEN // PR0
				RadExp_Step:=66;
			END_IF; 
			
		66:
			bSend:=FALSE;
	END_CASE
	
	SendStringS1(sSendStringS:= , bSendByte=> );
				Write_0.szSize:=INT_TO_USINT(LIMIT(0,LEN(SendStringS1.sSendStringS),10))+2;
				Write_0.pBuffer:=ADR(SendStringS1.bSendByte);
END_ACTION

ACTION _a_Init_active:
	
	CASE Init_Step OF 
		0:	//参数初始化
			bSend	 :=FALSE;
			Init_Step:=10;
			
		10:	//建立通讯
			SendStringS1.sSendStringS:='ST';
			bSend:=BLINK1_ST.OUT;  
			IF ReadString.RecvString='ST001' OR ReadString.RecvString='ST002' THEN //收到ST000，通讯正常//此版本是001，所有状态都加1，文档状态说明都加1
				Init_Step:=20;
			ELSE
				iAlarmNum:=301;		//通讯错误
			END_IF
			
		20://检查错误,如果有错误，就复位，没错误，延迟2秒跳转
			iAlarmNum:=0;		//通讯
			IF byReadData[0]= 16#45 AND (byReadData[1]= 16#4C) THEN //收到ER或EL,确认收到了错误信号，EL可以理解为可恢复，ER为不可恢复 收到EL信号可复位，ER信号只是显示
				SendStringS1.sSendStringS:=ReadString.RecvString;
				bSend:=BLINK1.OUT;
				TON3(IN:=FALSE);
			ELSE
				TON3(IN:=TRUE , PT:=T#2S);//2秒内无报错
				IF TON3.Q THEN
					SendStringS1.sSendStringS:='ST';
					bSend:=BLINK1.OUT;
					IF ReadString.RecvString='ST002' OR ReadString.RecvString='ST001' THEN //收到ST002，通讯正常//此版本是001，所有状态都加1
						Init_Step:=66;
					END_IF
				END_IF;
			END_IF
		66:
			;
		ELSE
			;
		END_CASE
		(*射线源状态*)
		GVL_State.iXray_State:=20;
		SendStringS1(sSendStringS:= , bSendByte=> );
		Write_0.szSize:=INT_TO_USINT(LIMIT(0,LEN(SendStringS1.sSendStringS),10))+2;
		Write_0.pBuffer:=ADR(SendStringS1.bSendByte);
		
		TON11(in:=FALSE);
END_ACTION

ACTION _QueryState_entry:
GVL_State.iXray_State:=40;

TON11(in:=FALSE);
END_ACTION

ACTION _Debug_active:

	IF (byReadData[0]=16#45 AND byReadData[1]=16#4C) OR (byReadData[0]=16#45 AND byReadData[1]=16#52) THEN // EL和ER 的错误
		ASCII_Chart_N_Alarm[3](byASCII:=byReadData[2] , sOut_Single=> );
		ASCII_Chart_N_Alarm[4](byASCII:=byReadData[3] , sOut_Single=> );
		ASCII_Chart_N_Alarm[5](byASCII:=byReadData[4] , sOut_Single=> );
		iAlarmNum:=STRING_TO_BYTE(ASCII_Chart_N_Alarm[3].sOut_Single)*100+STRING_TO_BYTE(ASCII_Chart_N_Alarm[4].sOut_Single)*10+STRING_TO_BYTE(ASCII_Chart_N_Alarm[5].sOut_Single);
		bXrayError1:=TRUE;
	ELSE
		bXrayError1	:=FALSE;
	//	iAlarmNum	:=0;
	END_IF

	TOF11(IN:= bXrayError1, PT:=T#5S , Q=>bXrayError , ET=> );
	
	IF bXrayError THEN
		GVL_State.iXray_State:=44;
	ELSE
		iAlarmNum	:=0;
	END_IF
	
	
	IF GVL_State.iXray_State<>40 THEN
		FOR k:=0 TO 30 BY 1 DO
			IF byReadData[k]=16#48 AND byReadData[k+1]=16#45 AND (byReadData[k+2]>=16#30 AND byReadData[k+2]<=16#39) THEN //保证是数字
				ASCII_Chart_N2[0](byASCII:= byReadData[k+2], sOut_Single=> );
				ASCII_Chart_N2[1](byASCII:= byReadData[k+3], sOut_Single=> );
				ASCII_Chart_N2[2](byASCII:= byReadData[k+4], sOut_Single=> );
				Feedback_nMHuValue:=STRING_TO_REAL(ASCII_Chart_N2[0].sOut_Single)*100+STRING_TO_REAL(ASCII_Chart_N2[1].sOut_Single)*10+STRING_TO_REAL(ASCII_Chart_N2[2].sOut_Single);
			END_IF
		END_FOR
	END_IF;

	IF (byReadData[0]=16#45 AND byReadData[1]=16#4C) THEN
		ASCII_Chart_N_Alarm1(byASCII:=	byReadData[2] , sOut_Single=> );
		ASCII_Chart_N_Alarm2(byASCII:= 	byReadData[3], sOut_Single=> );
		ASCII_Chart_N_Alarm3(byASCII:= 	byReadData[4], sOut_Single=> );
		sResetError1:=CONCAT('EL',ASCII_Chart_N_Alarm1.sOut_Single);
		sResetError2:=CONCAT(sResetError1,ASCII_Chart_N_Alarm2.sOut_Single);
		sResetError3:=CONCAT(sResetError2,ASCII_Chart_N_Alarm3.sOut_Single);
		SendStringS1.sSendStringS:=sResetError3;
	END_IF;
	
	IF bResetXray1 THEN
		SendStringS1(sSendStringS:= , bSendByte=> );
		Write_0.szSize:=INT_TO_USINT(LIMIT(0,LEN(SendStringS1.sSendStringS),10))+2;
		Write_0.pBuffer:=ADR(SendStringS1.bSendByte);
		bSend:=bResetXray1;
	END_IF
	
	IF bResetXray2 THEN
		byReadData[0]:=0;
	END_IF
(*	
	IF byReadData[0]=16#48 AND byReadData[1]=16#45 THEN 			//HE 球管热量
			ASCII_Chart_N2[0](byASCII:= byReadData[2], sOut_Single=> );
			ASCII_Chart_N2[1](byASCII:= byReadData[3], sOut_Single=> );
			ASCII_Chart_N2[2](byASCII:= byReadData[4], sOut_Single=> );
			Feedback_nMHuValue:=STRING_TO_REAL(ASCII_Chart_N2[0].sOut_Single)*100+STRING_TO_REAL(ASCII_Chart_N2[1].sOut_Single)*10+STRING_TO_REAL(ASCII_Chart_N2[2].sOut_Single);
		ELSE
			IF byReadData[8]=16#48 AND byReadData[9]=16#45 THEN 			//HE 球管热量
				ASCII_Chart_N2[0](byASCII:= byReadData[10], sOut_Single=> );
				ASCII_Chart_N2[1](byASCII:= byReadData[11], sOut_Single=> );
				ASCII_Chart_N2[2](byASCII:= byReadData[12], sOut_Single=> );
				Feedback_nMHuValue:=STRING_TO_REAL(ASCII_Chart_N2[0].sOut_Single)*100+STRING_TO_REAL(ASCII_Chart_N2[1].sOut_Single)*10+STRING_TO_REAL(ASCII_Chart_N2[2].sOut_Single);
			END_IF
		END_IF
	*)
END_ACTION

ACTION _Exposure1_entry:
bJumpRadExp:=false;
END_ACTION

ACTION _QueryState_active:

GVL_State.iXray_State:=40;
		CASE Query_Step OF 	
			//跳转后的中间变量复位工作
			0:
				bSend		:=FALSE;
			//	RadExp_Step	:=0;
			//	RadFlu_Step	:=0;
				Query_Step	:=10;
				ExpPara_Step:=0;
				FluPara_Setp:=0;
				DR_Para		:=0;
				
			10:
				(*1.查询命令*)
				CASE Lookup_Step OF 
					0:
						SendStringS1.sSendStringS:='ST';//当前状态
						IF BLINK1_ST.OUT THEN
							Lookup_Step:=1;
						END_IF
					1:
						SendStringS1.sSendStringS:='RR';//曝光模式下的查询
						IF NOT(BLINK1_ST.OUT) THEN
							Lookup_Step:=2;
						END_IF
					2:
						SendStringS1.sSendStringS:='RF';//透视模式下的查询
						IF BLINK1_ST.OUT THEN
							Lookup_Step:=3;
						END_IF
					3:
						SendStringS1.sSendStringS:='HE?';//球管热量
						IF NOT(BLINK1_ST.OUT) THEN
							Lookup_Step:=4;
						END_IF
					4:
						SendStringS1.sSendStringS:='FO?';//当前焦点
						IF BLINK1_ST.OUT THEN
							Lookup_Step:=5;
						END_IF
					5:
						SendStringS1.sSendStringS:='MS?';//曝光时间
						IF NOT(BLINK1_ST.OUT) THEN
							Lookup_Step:=0;
						END_IF
				END_CASE
				(*2.数据解析*)
				bSend:=BLINK1_1S.OUT;	//2秒查询一次	
				
				IF byReadData[0]=16#48 AND byReadData[1]=16#45 THEN 			//HE 球管热量
					ASCII_Chart_N2[0](byASCII:= byReadData[2], sOut_Single=> );
					ASCII_Chart_N2[1](byASCII:= byReadData[3], sOut_Single=> );
					ASCII_Chart_N2[2](byASCII:= byReadData[4], sOut_Single=> );
					Feedback_nMHuValue:=STRING_TO_REAL(ASCII_Chart_N2[0].sOut_Single)*100+STRING_TO_REAL(ASCII_Chart_N2[1].sOut_Single)*10+STRING_TO_REAL(ASCII_Chart_N2[2].sOut_Single);
				END_IF
				
				IF byReadData[0]=16#46 AND byReadData[1]=16#4C AND byReadData[2]=16#4B THEN //RF的FLK电压反馈
					ASCII_Chart_N2[0](byASCII:= byReadData[3], sOut_Single=> );
					ASCII_Chart_N2[1](byASCII:= byReadData[4], sOut_Single=> );
					ASCII_Chart_N2[2](byASCII:= byReadData[5], sOut_Single=> );
					Feedback_Kv:=STRING_TO_UDINT(ASCII_Chart_N2[0].sOut_Single)*100+STRING_TO_UDINT(ASCII_Chart_N2[1].sOut_Single)*10+STRING_TO_UDINT(ASCII_Chart_N2[2].sOut_Single);
				END_IF
				
				IF byReadData[7]=16#46 AND byReadData[8]=16#4C AND byReadData[9]=16#4D THEN //RF的FLM电流反馈
					ASCII_Chart_N2[0](byASCII:= byReadData[10], sOut_Single=> );
					ASCII_Chart_N2[1](byASCII:= byReadData[11], sOut_Single=> );
					ASCII_Chart_N2[2](byASCII:= byReadData[12], sOut_Single=> );
					Feedback_mA:=STRING_TO_REAL(ASCII_Chart_N2[0].sOut_Single)*10+STRING_TO_REAL(ASCII_Chart_N2[1].sOut_Single)*1+STRING_TO_REAL(ASCII_Chart_N2[2].sOut_Single)*0.1;
				END_IF

				IF byReadData[7]=16#46 AND byReadData[8]=16#4F THEN 					//FO的焦点反馈
					ASCII_Chart_N2[0](byASCII:= byReadData[2], sOut_Single=> );
					Feedback_nFocus:=STRING_TO_UDINT(ASCII_Chart_N2[2].sOut_Single);
				END_IF
			END_CASE
			
			SendStringS1(sSendStringS:= , bSendByte=> );
			Write_0.szSize:=INT_TO_USINT(LIMIT(0,LEN(SendStringS1.sSendStringS),10))+2;
			Write_0.pBuffer:=ADR(SendStringS1.bSendByte);
END_ACTION

ACTION _DefaultPara_entry:
GVL_State.iXray_State:=30;
END_ACTION

ACTION _DefaultPara_active:


		CASE Default_Step OF 
		0:
			bSend:=FALSE;
			Default_Step:=10;
	
		10://1.关闭AEC
			SendStringS1.sSendStringS:='FI000';
			bSend:=BLINK1.OUT;
			IF ReadString.RecvString=SendStringS1.sSendStringS THEN
				Default_Step:=20;
			END_IF
			
		20://EXPOSURE TECHNIQUE SELECTION
			SendStringS1.sSendStringS:='ET1';
			bSend:=BLINK1.OUT;
			IF ReadString.RecvString=SendStringS1.sSendStringS THEN
				Default_Step:=30;
			END_IF
			
		30:
			Default_Step:=66;
			bSend:=FALSE;
		ELSE 
			;
		END_CASE
		SendStringS1(sSendStringS:= , bSendByte=> );
		Write_0.szSize:=INT_TO_USINT(LIMIT(0,LEN(SendStringS1.sSendStringS),10))+2;
		Write_0.pBuffer:=ADR(SendStringS1.bSendByte);
END_ACTION

ACTION _a_DrExposure_active_1:


(*---------------------------曝光状态---------------------------------*)
			CASE DR_Step OF
				0:
					bSend:=FALSE;R_TRIG1(CLK:=FALSE);R_TRIG2(CLK:=FALSE);R_TRIG3(CLK:=FALSE);R_TRIG4(CLK:=FALSE);
					TON12(IN:=FALSE);TON13(IN:=FALSE);
					DR_Step:=5;
				
				5:
					TON12(IN:= Entity_IO.bXaryOne AND Entity_IO.bXaryTwo, PT:= T#3S, Q=> , ET=> );
					IF TON12.Q THEN
						DR_Step:=55;
					END_IF

				55:
					IF ReadString.RecvString='PR0' THEN // PR0
						SendStringS1.sSendStringS:='PR0';//曝光完成
						R_TRIG1(CLK:=ReadString.RecvString='PR0' , Q=>bSend );//收到立刻发送
						DR_Step:=66;
					END_IF;
					
				66:
					IF Entity_IO.bXaryOne=FALSE AND Entity_IO.bXaryTwo=FALSE THEN
						//IF ReadString.RecvString='PR0' THEN // PR0
						IF (byReadData[0]=16#50 AND byReadData[1]=16#52 AND byReadData[2]=16#30) THEN // PR0  规避字符串较长情况
							SendStringS1.sSendStringS:='PR0';//曝光完成
							bSend:=BLINK1.OUT;
							TON13(IN:=TRUE , PT:= T#2S, Q=> , ET=> );
						END_IF;
					END_IF;
					
					IF TON13.Q THEN
						DR_Step:=77;
					END_IF

				77:
					bSend:=FALSE;	
				END_CASE
			
				SendStringS1(sSendStringS:= , bSendByte=> );
				Write_0.szSize:=INT_TO_USINT(LIMIT(0,LEN(SendStringS1.sSendStringS),10))+2;
				Write_0.pBuffer:=ADR(SendStringS1.bSendByte);
END_ACTION

ACTION _a_DrExposure_entry_1:


DR_Step:=0;
GVL_State.iXray_State:=100;
END_ACTION

ACTION _a_DrPara_active_1:


	CASE DR_Para OF 
		0:
			IF GVL_State.iPLC_State=110 THEN //静态DR
				iDR_Staiton:=3;
			ELSIF GVL_State.iPLC_State=120 THEN //只有动态DR的时候，启动曝光触发
				iDR_Staiton:=4;
			ELSE
				iDR_Staiton:=3;
			END_IF;
		
			TOF_DR1(IN:=(Entity_IO.bXrayOneInput OR Entity_IO.bXayExpoInput) , PT:= T#500MS, Q=>, ET=> ); //按了一档，但此时没有输出1档给射线源
			IF TOF_DR1.Q THEN		
				(*大命令写入*)
				ExpParaSet(
							WS:= iDR_Staiton, //工作站
							FO:= UDINT_TO_UINT(WorkStation_TCP.PLC_RECV1.m_nFocus), //焦点
							ET:= 1, //AEC
							FI:= 0, //AEC
							FS:= 1,
							FN:= 0, //
							KV:= UDINT_TO_UINT(WorkStation_TCP.PLC_RECV1.m_nKv), //电压
							MA:= REAL_TO_UINT(WorkStation_TCP.PLC_RECV1.m_nMA*10), //电流
							MS:= REAL_TO_UINT(WorkStation_TCP.PLC_RECV1.m_nMS*10), //曝光时间
							Out=> );
								
				(*字符串存储到数组里*)			
					String_TO_ASCII1(
										InputString:=ExpParaSet.Out , 
										MaxArraySize:= 255, 
										ASCIIArray=> ArrASCII, 
										ArrayLength=> , 
										Error=> , 
										ErrorMessage=> );
														
				(*计算和校验*)		
					CheckSum:=0;
					FOR j:=1 TO 53 BY 1 DO
						IF ArrASCII[j]=16#0 THEN   	//空格对应的ASCII码不计入和校验中
							CONTINUE;
						END_IF
						CheckSum:=CheckSum+ArrASCII[j];
					END_FOR
					
				(*处理和校验，并转化成字符串形式*)
					CheckSum1:=CheckSum+16#03;
					CheckSum2:=(CheckSum1) AND 16#FF; 	//取低字节byte
					
					ArrASCII[54]:=3;
					ArrASCII[55]:=UINT_TO_BYTE(CheckSum2);
			
				(*发送指令*)	
					Write_0.szSize:=INT_TO_USINT(LIMIT(0,LEN(ExpParaSet.Out),255))+2;//获取写入的字符串长度	已增加03H结束符+CheckSum和校验
					Write_0.pBuffer:=ADR(ArrASCII);	
					bSend:=BLINK1.OUT;
					
					IF byReadData[0]=16#57 AND byReadData[1]=16#53 THEN //返回WS
						DR_Para:=20;
					END_IF;
			END_IF;
			
				
			10://Bucky处理
				IF GVL_State.iPLC_State=110 THEN //静态DR
					SendStringS1.sSendStringS:='BU0';
				ELSIF GVL_State.iPLC_State=120 THEN //只有动态DR的时候，启动曝光触发
					SendStringS1.sSendStringS:='BU1';
				END_IF;
				
				bSend:=BLINK1.OUT;
				IF ReadString.RecvString=SendStringS1.sSendStringS THEN
					ExpPara_Step:=20;
				END_IF
				SendStringS1(sSendStringS:= , bSendByte=> );
				Write_0.szSize:=INT_TO_USINT(LIMIT(0,LEN(SendStringS1.sSendStringS),10))+2;
				Write_0.pBuffer:=ADR(SendStringS1.bSendByte);
				
			20:
				DR_Para:=66;
	END_CASE
END_ACTION

ACTION _a_DrPara_entry_1:


DR_Para:=0;
GVL_State.iXray_State:=90;
END_ACTION

ACTION _a_FluoroPara_active_1:


	CASE FluPara_Setp OF 
		0:
		(*大命令写入*)
			FluParaSet(
						WS:= 2, //工作站
						FLF:= 2, //脉冲透视
						FLA:= 0, //不使用ABS
						FLS:= 170, //脉冲透视频率×10//1114
						FLR:= 1, //透视累计时间清零
						FLK:= UDINT_TO_UINT(WorkStation_TCP.PLC_RECV1.m_nKv), //透视电压
						FLM:= REAL_TO_UINT(WorkStation_TCP.PLC_RECV1.m_nMA*10),//透视电流×10
						Out=> );
						
		(*字符串存储到数组里*)			
			String_TO_ASCII1(
								InputString:=FluParaSet.Out , 
								MaxArraySize:= 255, 
								ASCIIArray=> ArrASCII, 
								ArrayLength=> , 
								Error=> , 
								ErrorMessage=> );
								
					
		(*计算和校验*)		
			CheckSum:=0;
			FOR j:=1 TO 43 BY 1 DO
				IF ArrASCII[j]=16#00 THEN   	//空格对应的ASCII码不计入和校验中
					CONTINUE;
				END_IF
				CheckSum:=CheckSum+ArrASCII[j];
			END_FOR
			
			(*处理和校验，并转化成字符串形式*)
			CheckSum3:=CheckSum+16#03;
			CheckSum4:=(CheckSum3) AND 16#FF; 	//取低字节byte
			
			ArrASCII[44]:=3;
			ArrASCII[45]:=UINT_TO_BYTE(CheckSum4);
	
		(*发送指令*)	
			Write_0.szSize:=INT_TO_USINT(LIMIT(0,LEN(FluParaSet.Out),255))+2;//获取写入的字符串长度	已增加03H结束符+CheckSum和校验
			Write_0.pBuffer:=ADR(ArrASCII);	
			bSend:=BLINK1.OUT;
			
			IF byReadData[0]=16#57 AND byReadData[1]=16#53 THEN //返回WS
				FluPara_Setp:=10;
			END_IF;
	
		10:
			FluPara_Setp:=66;

	END_CASE
END_ACTION

ACTION _a_FluoroPara_entry_1:

FluPara_Setp:=0;
GVL_State.iXray_State:=70;
RadFlu_Step	:=0;
END_ACTION

ACTION _a_FluoroExPosure_active_1:


		(*---------------------------曝光状态---------------------------------*)
			CASE RadFlu_Step OF
				0:	//透视信号给定
					IF ReadString.RecvString='FLP1' THEN
						RadFlu_Step	:=10;
					END_IF;	
					
					IF ReadString.RecvString='FLX0' OR ReadString.RecvString='FLP0' OR  ReadString.RecvString='FLFLX0'  OR  ReadString.RecvString='FLFLP0' THEN //收到FLX0或FLP0，曝光结束
						RadFlu_Step	:=30;
					END_IF;	
					
				10://FLX1 脉冲信号给定
					IF ReadString.RecvString='FLX1' THEN
						RadFlu_Step	:=20;
					END_IF;
					
					IF ReadString.RecvString='FLX0' OR ReadString.RecvString='FLP0' OR  ReadString.RecvString='FLFLX0'  OR  ReadString.RecvString='FLFLP0' THEN //收到FLX0或FLP0，曝光结束
						RadFlu_Step	:=30;
					END_IF;	
					
				20://出束阶段
					IF ReadString.RecvString='FLX0' OR ReadString.RecvString='FLP0' OR  ReadString.RecvString='FLFLX0'  OR  ReadString.RecvString='FLFLP0' THEN //收到FLX0或FLP0，曝光结束 THEN 增加了一个字符串位的情况
						RadFlu_Step	:=66;
					ELSE
						;
					END_IF
					
				 30://结束
					RadFlu_Step	:=66;
				
				66:
					;
				ELSE
					;
				END_CASE
END_ACTION

ACTION _a_FluoroExPosure_entry_1:

TON_HangOver(IN:=FALSE);
RadFlu_Step:=0;
GVL_State.iXray_State:=80;
END_ACTION

ACTION _a_ExposurePara_active_1:

(**此程序未考虑，DR模式*)
CASE ExpPara_Step OF 
		0:
		(*大命令写入*)
		ExpParaSet(
					WS:= 1, //工作站
					FO:= UDINT_TO_UINT(WorkStation_TCP.PLC_RECV1.m_nFocus), //焦点
					ET:= 1, //AEC
					FI:= 0, //AEC
					FS:= 1,
					FN:= 0, //
					KV:= UDINT_TO_UINT(WorkStation_TCP.PLC_RECV1.m_nKv), //电压
					MA:= REAL_TO_UINT(WorkStation_TCP.PLC_RECV1.m_nMA*10), //电流
					MS:= REAL_TO_UINT(WorkStation_TCP.PLC_RECV1.m_nMS*10), //曝光时间
					Out=> );
						
		(*字符串存储到数组里*)			
			String_TO_ASCII1(
								InputString:=ExpParaSet.Out , 
								MaxArraySize:= 255, 
								ASCIIArray=> ArrASCII, 
								ArrayLength=> , 
								Error=> , 
								ErrorMessage=> );
												
		(*计算和校验*)		
			CheckSum:=0;
			FOR j:=1 TO 53 BY 1 DO
				IF ArrASCII[j]=16#0 THEN   	//空格对应的ASCII码不计入和校验中
					CONTINUE;
				END_IF
				CheckSum:=CheckSum+ArrASCII[j];
			END_FOR
			
		(*处理和校验，并转化成字符串形式*)
			CheckSum1:=CheckSum+16#03;
			CheckSum2:=(CheckSum1) AND 16#FF; 	//取低字节byte
			
			ArrASCII[54]:=3;
			ArrASCII[55]:=UINT_TO_BYTE(CheckSum2);
	
		(*发送指令*)	
			Write_0.szSize:=INT_TO_USINT(LIMIT(0,LEN(ExpParaSet.Out),255))+2;//获取写入的字符串长度	已增加03H结束符+CheckSum和校验
			Write_0.pBuffer:=ADR(ArrASCII);	
			bSend:=BLINK1.OUT;
			
			IF byReadData[0]=16#57 AND byReadData[1]=16#53 THEN //返回WS
				ExpPara_Step:=20;
			END_IF;
			
		10://Bucky处理
			IF GVL_State.iPLC_State=210 OR GVL_State.iPLC_State=220 OR GVL_State.iPLC_State=240 THEN
				SendStringS1.sSendStringS:='BU0';
			ELSIF GVL_State.iPLC_State=120 THEN 			//只有动态DR的时候，启动曝光触发
				SendStringS1.sSendStringS:='BU1';
			END_IF;
			
			bSend:=BLINK1.OUT;
			IF ReadString.RecvString=SendStringS1.sSendStringS THEN
				ExpPara_Step:=20;
			END_IF
			SendStringS1(sSendStringS:= , bSendByte=> );
			Write_0.szSize:=INT_TO_USINT(LIMIT(0,LEN(SendStringS1.sSendStringS),10))+2;
			Write_0.pBuffer:=ADR(SendStringS1.bSendByte);
			
		20:
			ExpPara_Step:=66;
	END_CASE
END_ACTION

ACTION _a_ExposurePara_entry_1:
	ExpPara_Step:=0;
	GVL_State.iXray_State:=50;
END_ACTION

ACTION _a_Exposure_active_1:


	(*---------------------------曝光状态---------------------------------*)
			CASE RadExp_Step OF
				0:
					bSend:=FALSE;R_TRIG1(CLK:=FALSE);R_TRIG2(CLK:=FALSE);R_TRIG3(CLK:=FALSE);R_TRIG4(CLK:=FALSE);
					TON12(IN:=FALSE);TON13(IN:=FALSE);
					RadExp_Step:=5;
					
				5:
					TON12(IN:= Entity_IO.bXaryOne AND Entity_IO.bXaryTwo, PT:= T#3S, Q=> , ET=> );
					IF TON12.Q THEN
						RadExp_Step:=55;
					END_IF

				55:
					SendStringS1.sSendStringS:='PR0';
					IF ReadString.RecvString='PR0' THEN // PR0
						R_TRIG1(CLK:=ReadString.RecvString='PR0' , Q=>bSend );	//收到立刻发送
						RadExp_Step:=66;
					END_IF;
					
						
				66:
					SendStringS1.sSendStringS:='PR0';
					IF Entity_IO.bXaryOne=FALSE AND Entity_IO.bXaryTwo=FALSE THEN
						//IF ReadString.RecvString='PR0' THEN // PR0
						IF (byReadData[0]=16#50 AND byReadData[1]=16#52 AND byReadData[2]=16#30) THEN // PR0  规避字符串较长情况
							bSend:=BLINK1.OUT;
							TON13(IN:=TRUE , PT:= T#2S, Q=> , ET=> );
						END_IF;
					END_IF;
					
					IF TON13.Q THEN
						RadExp_Step:=77;
					END_IF
					
				77:
					bSend:=FALSE;
			
			END_CASE
				SendStringS1(sSendStringS:= , bSendByte=> );
				Write_0.szSize:=INT_TO_USINT(LIMIT(0,LEN(SendStringS1.sSendStringS),10))+2;
				Write_0.pBuffer:=ADR(SendStringS1.bSendByte);
END_ACTION

ACTION _a_Exposure_entry_1:
	RadExp_Step:=0;
	GVL_State.iXray_State:=60;
	bSend:=FALSE;
END_ACTION

ACTION _Error_entry:
	

	Step_Error:=0;
END_ACTION

ACTION _QueryState_exit:

	Query_Step:=0;
END_ACTION

ACTION _a_FluoroExPosure_exit:
FluPara_Setp:=0;
END_ACTION

END_PROGRAM

// Device/Application/aSpecailBasic/RecvStringS
FUNCTION_BLOCK RecvStringS 
VAR_INPUT
	Excute:BOOL;
	Size:INT;
	RecvArray:ARRAY [0..255] OF BYTE;
END_VAR
VAR_OUTPUT
	RecvString:STRING;
END_VAR
VAR
	i,j:INT;
	RecvNum:INT;
	R_TRIG1:R_TRIG;
	sRecvArray:ARRAY [0..255] OF STRING;
	ASCII_Chart_N1:ARRAY [0..255] OF ASCII_Chart_N;
END_VAR

//readme
//1.单命令解析
//2.单命令最多8个字符

	R_TRIG1(CLK:=Excute, Q=> );		//获取读到了多少个字符
	IF R_TRIG1.Q THEN
		RecvNum:=LIMIT(0,Size-2,9);	//减去结束位和校验位
	END_IF;

	FOR i:=0 TO RecvNum BY 1 DO 
		ASCII_Chart_N1[i](byASCII:=RecvArray[i] , sOut_Single=>sRecvArray[i] );//调用单字符输出
	END_FOR 
	
	RecvString :='';
	FOR i := 0 TO RecvNum-1 DO
    	RecvString := CONCAT(RecvString, sRecvArray[i]);  // 循环拼接数组元素
	END_FOR;

END_FUNCTION_BLOCK

// Device/Application/BasicFBs/ASCII_Chart_N
FUNCTION_BLOCK ASCII_Chart_N
VAR_INPUT
	byASCII		:BYTE;
END_VAR
VAR_OUTPUT
	sOut_Single	:STRING;
END_VAR
VAR
	
END_VAR

(*ASCII码转化为字符*)
	
	IF    byASCII=16#41 THEN 	sOut_Single:='A';
	ELSIF byASCII=16#42 THEN  	sOut_Single:='B';
	ELSIF byASCII=16#43 THEN  	sOut_Single:='C';
	ELSIF byASCII=16#44 THEN	sOut_Single:='D';
	ELSIF byASCII=16#45 THEN	sOut_Single:='E';
	ELSIF byASCII=16#46 THEN	sOut_Single:='F';
	ELSIF byASCII=16#47 THEN	sOut_Single:='G';
	ELSIF byASCII=16#48 THEN	sOut_Single:='H';
	ELSIF byASCII=16#49 THEN	sOut_Single:='I';
	ELSIF byASCII=16#4A THEN	sOut_Single:='J';
	ELSIF byASCII=16#4B THEN	sOut_Single:='K';
	ELSIF byASCII=16#4C THEN	sOut_Single:='L';
	ELSIF byASCII=16#4D THEN	sOut_Single:='M';
	ELSIF byASCII=16#4E THEN	sOut_Single:='N';
	ELSIF byASCII=16#4F THEN	sOut_Single:='O';
	ELSIF byASCII=16#50 THEN	sOut_Single:='P';
	ELSIF byASCII=16#51 THEN	sOut_Single:='Q';
	ELSIF byASCII=16#52 THEN	sOut_Single:='R';
	ELSIF byASCII=16#53 THEN	sOut_Single:='S';
	ELSIF byASCII=16#54 THEN	sOut_Single:='T';
	ELSIF byASCII=16#55 THEN	sOut_Single:='U';
	ELSIF byASCII=16#56 THEN	sOut_Single:='V';
	ELSIF byASCII=16#57 THEN	sOut_Single:='W';
	ELSIF byASCII=16#58 THEN	sOut_Single:='X';
	ELSIF byASCII=16#59 THEN	sOut_Single:='Y';
	ELSIF byASCII=16#5A THEN	sOut_Single:='Z';
	ELSIF byASCII=16#5B THEN	sOut_Single:='[';
	ELSIF byASCII=16#5C THEN	sOut_Single:='\';
	ELSIF byASCII=16#5D THEN	sOut_Single:=']';
	ELSIF byASCII=16#5E THEN	sOut_Single:='^';
	ELSIF byASCII=16#5F THEN	sOut_Single:='_';
	ELSIF byASCII=16#60 THEN	sOut_Single:='`';
	                                         
	ELSIF byASCII=16#61 THEN	sOut_Single:='a';
	ELSIF byASCII=16#62 THEN  	sOut_Single:='b';
	ELSIF byASCII=16#63 THEN  	sOut_Single:='c';
	ELSIF byASCII=16#64 THEN	sOut_Single:='d';
	ELSIF byASCII=16#65 THEN	sOut_Single:='e';
	ELSIF byASCII=16#66 THEN	sOut_Single:='f';
	ELSIF byASCII=16#67 THEN	sOut_Single:='g';
	ELSIF byASCII=16#68 THEN	sOut_Single:='h';
	ELSIF byASCII=16#69 THEN	sOut_Single:='i';
	ELSIF byASCII=16#6A THEN	sOut_Single:='j';
	ELSIF byASCII=16#6B THEN	sOut_Single:='k';
	ELSIF byASCII=16#6C THEN	sOut_Single:='l';
	ELSIF byASCII=16#6D THEN	sOut_Single:='m';
	ELSIF byASCII=16#6E THEN	sOut_Single:='n';
	ELSIF byASCII=16#6F THEN	sOut_Single:='o';
	ELSIF byASCII=16#70 THEN	sOut_Single:='p';
	ELSIF byASCII=16#71 THEN	sOut_Single:='q';
	ELSIF byASCII=16#72 THEN	sOut_Single:='r';
	ELSIF byASCII=16#73 THEN	sOut_Single:='s';
	ELSIF byASCII=16#74 THEN	sOut_Single:='t';
	ELSIF byASCII=16#75 THEN	sOut_Single:='u';
	ELSIF byASCII=16#76 THEN	sOut_Single:='v';
	ELSIF byASCII=16#77 THEN	sOut_Single:='w';
	ELSIF byASCII=16#78 THEN	sOut_Single:='x';
	ELSIF byASCII=16#79 THEN	sOut_Single:='y';
	ELSIF byASCII=16#7A THEN	sOut_Single:='z';
	ELSIF byASCII=16#7B THEN	sOut_Single:='{';
	ELSIF byASCII=16#7C THEN	sOut_Single:='|';
	ELSIF byASCII=16#7D THEN	sOut_Single:='}';
	                                         
	ELSIF byASCII=16#30 THEN  	sOut_Single:='0';
	ELSIF byASCII=16#31 THEN  	sOut_Single:='1';
	ELSIF byASCII=16#32 THEN	sOut_Single:='2';
	ELSIF byASCII=16#33 THEN	sOut_Single:='3';
	ELSIF byASCII=16#34 THEN	sOut_Single:='4';
	ELSIF byASCII=16#35 THEN	sOut_Single:='5';
	ELSIF byASCII=16#36 THEN	sOut_Single:='6';
	ELSIF byASCII=16#37 THEN	sOut_Single:='7';
	ELSIF byASCII=16#38 THEN	sOut_Single:='8';
	ELSIF byASCII=16#39 THEN	sOut_Single:='9';
	ELSIF byASCII=16#3A THEN	sOut_Single:=':';
	ELSIF byASCII=16#3B THEN	sOut_Single:=';';
	ELSIF byASCII=16#3C THEN	sOut_Single:='<';
	ELSIF byASCII=16#3D THEN	sOut_Single:='=';
	ELSIF byASCII=16#3E THEN	sOut_Single:='>';
	ELSIF byASCII=16#3F THEN	sOut_Single:='?';
	ELSIF byASCII=16#40 THEN	sOut_Single:='@';
	
	ELSIF byASCII=16#20 THEN	sOut_Single:=' ';	                                     
	ELSIF byASCII=16#21 THEN	sOut_Single:='!';
	ELSIF byASCII=16#22 THEN	sOut_Single:='"';
	ELSIF byASCII=16#23 THEN	sOut_Single:='#';
//	ELSIF byASCII=16#24 THEN	sOut_Single:='$';
	ELSIF byASCII=16#25 THEN	sOut_Single:='%';
	ELSIF byASCII=16#26 THEN	sOut_Single:='&';
//	ELSIF byASCII=16#27 THEN	sOut_Single:=''';
	ELSIF byASCII=16#28 THEN	sOut_Single:='(';
	ELSIF byASCII=16#29 THEN	sOut_Single:=')';
	ELSIF byASCII=16#2A THEN	sOut_Single:='*';
	ELSIF byASCII=16#2B THEN	sOut_Single:='+';
	ELSIF byASCII=16#2C THEN	sOut_Single:=',';
	ELSIF byASCII=16#2D THEN	sOut_Single:='-';
	ELSIF byASCII=16#2E THEN	sOut_Single:='.';
	ELSIF byASCII=16#2F THEN	sOut_Single:='/';
	ELSE
		;	 //错误标志
	END_IF

END_FUNCTION_BLOCK

// Device/Application/BasicFBs/Blink
FUNCTION_BLOCK Blink
(* Function block to simulate a turn signal *)
VAR_INPUT
	ENABLE:BOOL;		(* TRUE:run Blink, FALSE: OUT keeps its value*)
	TIMELOW:TIME;		(* Time for OUT=FALSE *)
	TIMEHIGH:TIME;		(* Time for OUT=TRUE *)
END_VAR
VAR_OUTPUT
	OUT:BOOL;			(* output variable, starting with FALSE *)
END_VAR
VAR
	CLOCK:TP;
END_VAR

(*======================== READ_ME ==============================*)
(*功能块：“闪烁”                                               *)
(***输出周期和占空比一定的矩形波                                 *)
(*=========================== END ===============================*)
		CLOCK( );							
	IF CLOCK.Q=FALSE AND ENABLE THEN			
		CLOCK(IN:=FALSE);							
		IF OUT=FALSE THEN
			CLOCK.PT:=TIMEHIGH;
		ELSE
			CLOCK.PT:=TIMELOW;
		END_IF;
		OUT := NOT OUT;									
		CLOCK(IN:=TRUE);
	ELSIF ENABLE=0 THEN	
		OUT :=0;					
	END_IF;

END_FUNCTION_BLOCK

// Device/Application/aSpecailBasic/SendStringS
FUNCTION_BLOCK SendStringS
VAR_INPUT
	sSendStringS:STRING;
END_VAR
VAR_OUTPUT
	bSendByte:ARRAY [0..255] OF BYTE;
END_VAR
VAR
	i:INT;
	iSize:INT;
	String2Byte1:String2Byte;
END_VAR



	iSize:=LIMIT(0,LEN(sSendStringS),10); 		//获取写入的字符串长度	已增加03H结束符+CheckSum和校验	
	String2Byte1(sXrayString:=sSendStringS , sByte=> );
//	Write_0.szSize:=INT_TO_USINT(iSize)+2;

	CASE iSize OF 
	2:
		(*2个字符的命令*)	
		bSendByte[0]:=String2Byte1.sByte[1];
		bSendByte[1]:=String2Byte1.sByte[2];
		bSendByte[2]:=16#03;
		bSendByte[3]:=bSendByte[0]+bSendByte[1]+bSendByte[2];
//		Write_0.pBuffer:=ADR(bSendByte);
	3:	
		(*3个字符的命令*)	
		bSendByte[0]:=String2Byte1.sByte[1];
		bSendByte[1]:=String2Byte1.sByte[2];
		bSendByte[2]:=String2Byte1.sByte[3];
		bSendByte[3]:=16#03;
		bSendByte[4]:=bSendByte[0]+bSendByte[1]+bSendByte[2]+bSendByte[3];
//		Write_0.pBuffer:=ADR(bSendByte);
	
	4:
		(*4个字符的命令*)	
		bSendByte[0]:=String2Byte1.sByte[1];
		bSendByte[1]:=String2Byte1.sByte[2];
		bSendByte[2]:=String2Byte1.sByte[3];
		bSendByte[3]:=String2Byte1.sByte[4];
		bSendByte[4]:=16#03;
		bSendByte[5]:=bSendByte[0]+bSendByte[1]+bSendByte[2]+bSendByte[3]+bSendByte[4];
//		Write_0.pBuffer:=ADR(bSendByte);
	
	5:
		(*5个字符的命令*)	
		bSendByte[0]:=String2Byte1.sByte[1];
		bSendByte[1]:=String2Byte1.sByte[2];
		bSendByte[2]:=String2Byte1.sByte[3];
		bSendByte[3]:=String2Byte1.sByte[4];
		bSendByte[4]:=String2Byte1.sByte[5];
		bSendByte[5]:=16#03;
		bSendByte[6]:=bSendByte[0]+bSendByte[1]+bSendByte[2]+bSendByte[3]+bSendByte[4]+bSendByte[5];
//		Write_0.pBuffer:=ADR(bSendByte);
		
	6:
		(*6个字符的命令*)	
		bSendByte[0]:=String2Byte1.sByte[1];
		bSendByte[1]:=String2Byte1.sByte[2];
		bSendByte[2]:=String2Byte1.sByte[3];
		bSendByte[3]:=String2Byte1.sByte[4];
		bSendByte[4]:=String2Byte1.sByte[5];
		bSendByte[5]:=String2Byte1.sByte[6];
		bSendByte[6]:=16#03;
		bSendByte[7]:=bSendByte[0]+bSendByte[1]+bSendByte[2]+bSendByte[3]+bSendByte[4]+bSendByte[5]+bSendByte[6];
//		Write_0.pBuffer:=ADR(bSendByte);		
	7:
		(*7个字符的命令*)	
		bSendByte[0]:=String2Byte1.sByte[1];
		bSendByte[1]:=String2Byte1.sByte[2];
		bSendByte[2]:=String2Byte1.sByte[3];
		bSendByte[3]:=String2Byte1.sByte[4];
		bSendByte[4]:=String2Byte1.sByte[5];
		bSendByte[5]:=String2Byte1.sByte[6];
		bSendByte[6]:=String2Byte1.sByte[7];
		bSendByte[7]:=16#03;
		bSendByte[8]:=bSendByte[0]+bSendByte[1]+bSendByte[2]+bSendByte[3]+bSendByte[4]+bSendByte[5]+bSendByte[6]+bSendByte[7];
//		Write_0.pBuffer:=ADR(bSendByte);
		
	8:(*8个字符的命令*)	
		bSendByte[0]:=String2Byte1.sByte[1];
		bSendByte[1]:=String2Byte1.sByte[2];
		bSendByte[2]:=String2Byte1.sByte[3];
		bSendByte[3]:=String2Byte1.sByte[4];
		bSendByte[4]:=String2Byte1.sByte[5];
		bSendByte[5]:=String2Byte1.sByte[6];
		bSendByte[6]:=String2Byte1.sByte[7];
		bSendByte[7]:=String2Byte1.sByte[8];
		bSendByte[8]:=16#03;
		bSendByte[9]:=bSendByte[0]+bSendByte[1]+bSendByte[2]+bSendByte[3]+bSendByte[4]+bSendByte[5]+bSendByte[6]+bSendByte[7]+bSendByte[8];
//		Write_0.pBuffer:=ADR(bSendByte);
	ELSE
		;//输入错误
	END_CASE

END_FUNCTION_BLOCK

// Device/Application/BasicFBs/String2Byte
FUNCTION_BLOCK String2Byte
VAR_INPUT
	 sXrayString:STRING;
END_VAR
VAR_OUTPUT
	 sByte	:ARRAY[0..9] OF BYTE;
END_VAR
VAR
	iSize	:INT;
	k		:INT:=1;
	s1		:STRING;
	sString	:ARRAY[0..9] OF STRING;
	ASCII_Chart1:ASCII_Chart_P;
END_VAR



	iSize:=LIMIT(0,LEN(sXrayString),10); //获取字符串长度
	
	(*获取每个字符，并放入字符序列中*)
	FOR k:=0 TO iSize BY 1 DO 
		s1:=MID(STR:= sXrayString, LEN:=1 , POS:=k );
		sString[k]:=s1;
		ASCII_Chart1(sASCII_IN:=s1 , byASCII=>sByte[k] );
	END_FOR

END_FUNCTION_BLOCK

// Device/Application/BasicFBs/ASCII_Chart_P
FUNCTION_BLOCK ASCII_Chart_P
VAR_INPUT
	sASCII_IN:STRING;
END_VAR
VAR_OUTPUT
	byASCII:BYTE;
END_VAR
VAR
	sIn_Single:STRING;
	
END_VAR

(*字符转换为16进制数字，BYTE数据类型*)

	sIn_Single:=LEFT(STR:=sASCII_IN , SIZE:=1 );//保证就一个字符
	
	IF    sIn_Single='A' THEN 	byASCII:=16#41;
	ELSIF sIn_Single='B' THEN  	byASCII:=16#42;
	ELSIF sIn_Single='C' THEN  	byASCII:=16#43;
	ELSIF sIn_Single='D' THEN	byASCII:=16#44;
	ELSIF sIn_Single='E' THEN	byASCII:=16#45;
	ELSIF sIn_Single='F' THEN	byASCII:=16#46;
	ELSIF sIn_Single='G' THEN	byASCII:=16#47;
	ELSIF sIn_Single='H' THEN	byASCII:=16#48;
	ELSIF sIn_Single='I' THEN	byASCII:=16#49;
	ELSIF sIn_Single='J' THEN	byASCII:=16#4A;
	ELSIF sIn_Single='K' THEN	byASCII:=16#4B;
	ELSIF sIn_Single='L' THEN	byASCII:=16#4C;
	ELSIF sIn_Single='M' THEN	byASCII:=16#4D;
	ELSIF sIn_Single='N' THEN	byASCII:=16#4E;
	ELSIF sIn_Single='O' THEN	byASCII:=16#4F;
	ELSIF sIn_Single='P' THEN	byASCII:=16#50;
	ELSIF sIn_Single='Q' THEN	byASCII:=16#51;
	ELSIF sIn_Single='R' THEN	byASCII:=16#52;
	ELSIF sIn_Single='S' THEN	byASCII:=16#53;
	ELSIF sIn_Single='T' THEN	byASCII:=16#54;
	ELSIF sIn_Single='U' THEN	byASCII:=16#55;
	ELSIF sIn_Single='V' THEN	byASCII:=16#56;
	ELSIF sIn_Single='W' THEN	byASCII:=16#57;
	ELSIF sIn_Single='X' THEN	byASCII:=16#58;
	ELSIF sIn_Single='Y' THEN	byASCII:=16#59;
	ELSIF sIn_Single='Z' THEN	byASCII:=16#5A;
	ELSIF sIn_Single='[' THEN	byASCII:=16#5B;
	ELSIF sIn_Single='\' THEN	byASCII:=16#5C;
	ELSIF sIn_Single=']' THEN	byASCII:=16#5D;
	ELSIF sIn_Single='^' THEN	byASCII:=16#5E;
	ELSIF sIn_Single='_' THEN	byASCII:=16#5F;
	ELSIF sIn_Single='`' THEN	byASCII:=16#60;
	
	ELSIF sIn_Single='a' THEN	byASCII:=16#61;	
	ELSIF sIn_Single='b' THEN  	byASCII:=16#62;
	ELSIF sIn_Single='c' THEN  	byASCII:=16#63;
	ELSIF sIn_Single='d' THEN	byASCII:=16#64;
	ELSIF sIn_Single='e' THEN	byASCII:=16#65;
	ELSIF sIn_Single='f' THEN	byASCII:=16#66;
	ELSIF sIn_Single='g' THEN	byASCII:=16#67;
	ELSIF sIn_Single='h' THEN	byASCII:=16#68;
	ELSIF sIn_Single='i' THEN	byASCII:=16#69;
	ELSIF sIn_Single='j' THEN	byASCII:=16#6A;
	ELSIF sIn_Single='k' THEN	byASCII:=16#6B;
	ELSIF sIn_Single='l' THEN	byASCII:=16#6C;
	ELSIF sIn_Single='m' THEN	byASCII:=16#6D;
	ELSIF sIn_Single='n' THEN	byASCII:=16#6E;
	ELSIF sIn_Single='o' THEN	byASCII:=16#6F;
	ELSIF sIn_Single='p' THEN	byASCII:=16#70;
	ELSIF sIn_Single='q' THEN	byASCII:=16#71;
	ELSIF sIn_Single='r' THEN	byASCII:=16#72;
	ELSIF sIn_Single='s' THEN	byASCII:=16#73;
	ELSIF sIn_Single='t' THEN	byASCII:=16#74;
	ELSIF sIn_Single='u' THEN	byASCII:=16#75;
	ELSIF sIn_Single='v' THEN	byASCII:=16#76;
	ELSIF sIn_Single='w' THEN	byASCII:=16#77;
	ELSIF sIn_Single='x' THEN	byASCII:=16#78;
	ELSIF sIn_Single='y' THEN	byASCII:=16#79;
	ELSIF sIn_Single='z' THEN	byASCII:=16#7A;
	ELSIF sIn_Single='{' THEN	byASCII:=16#7B;
	ELSIF sIn_Single='|' THEN	byASCII:=16#7C;
	ELSIF sIn_Single='}' THEN	byASCII:=16#7D;
	
	ELSIF sIn_Single='0' THEN  	byASCII:=16#30;
	ELSIF sIn_Single='1' THEN  	byASCII:=16#31;
	ELSIF sIn_Single='2' THEN	byASCII:=16#32;
	ELSIF sIn_Single='3' THEN	byASCII:=16#33;
	ELSIF sIn_Single='4' THEN	byASCII:=16#34;
	ELSIF sIn_Single='5' THEN	byASCII:=16#35;
	ELSIF sIn_Single='6' THEN	byASCII:=16#36;
	ELSIF sIn_Single='7' THEN	byASCII:=16#37;
	ELSIF sIn_Single='8' THEN	byASCII:=16#38;
	ELSIF sIn_Single='9' THEN	byASCII:=16#39;
	ELSIF sIn_Single=':' THEN	byASCII:=16#3A;
	ELSIF sIn_Single=';' THEN	byASCII:=16#3B;
	ELSIF sIn_Single='<' THEN	byASCII:=16#3C;
	ELSIF sIn_Single='=' THEN	byASCII:=16#3D;
	ELSIF sIn_Single='>' THEN	byASCII:=16#3E;
	ELSIF sIn_Single='?' THEN	byASCII:=16#3F;
	ELSIF sIn_Single='@' THEN	byASCII:=16#40;
		
	ELSIF sIn_Single=' ' THEN	byASCII:=16#20;
	ELSIF sIn_Single='!' THEN	byASCII:=16#21;
	ELSIF sIn_Single='"' THEN	byASCII:=16#22;
	ELSIF sIn_Single='#' THEN	byASCII:=16#23;
//	ELSIF sIn_Single='$' THEN	byASCII:=16#24;
	ELSIF sIn_Single='%' THEN	byASCII:=16#25;
	ELSIF sIn_Single='&' THEN	byASCII:=16#26;
//	ELSIF sIn_Single=''' THEN	byASCII:=16#27;
	ELSIF sIn_Single='(' THEN	byASCII:=16#28;
	ELSIF sIn_Single=')' THEN	byASCII:=16#29;
	ELSIF sIn_Single='*' THEN	byASCII:=16#2A;
	ELSIF sIn_Single='+' THEN	byASCII:=16#2B;
	ELSIF sIn_Single=',' THEN	byASCII:=16#2C;
	ELSIF sIn_Single='-' THEN	byASCII:=16#2D;
	ELSIF sIn_Single='.' THEN	byASCII:=16#2E;
	ELSIF sIn_Single='/' THEN	byASCII:=16#2F;
	ELSE
		byASCII:=16#FF;	 //错误标志
	END_IF

END_FUNCTION_BLOCK

// Device/Application/aSpecailBasic/X_RayFluPara
FUNCTION_BLOCK X_RayFluPara
VAR_INPUT

	WS:UINT;
	FLF:UINT;
	FLA:UINT;
	FLS:UINT;
	FLR:UINT;
	FLK:UINT;
	FLM:UINT;
	
END_VAR
VAR_OUTPUT
	Out:STRING;
END_VAR
VAR
	sString :ARRAY [0..15] OF STRING;
	sWString :ARRAY [0..15] OF STRING;
	
	sFLS,sFLK,sFLM:STRING;
END_VAR

(*Readme*)
(*透视模式下大命令组合命令*)

	sString[0]:=CONCAT(STR1:='FLU' , STR2:= ' ');
	
	sString[1]:=CONCAT(STR1:='WS' , STR2:= UINT_TO_STRING(WS));
	sString[2]:=CONCAT(STR1:=sString[1] ,STR2:= ' ');
	
	sString[3]:=CONCAT(STR1:='FLF' , STR2:= UINT_TO_STRING(FLF));
	sString[4]:=CONCAT(STR1:=sString[3] ,STR2:= ' ');
	
	sString[5]:=CONCAT(STR1:='FLA' , STR2:= UINT_TO_STRING(FLA));
	sString[6]:=CONCAT(STR1:=sString[5] ,STR2:= ' ');
	
	CASE FLS OF 
	0..9:
		sFLS:=CONCAT(STR1:='FLS00' , STR2:= UINT_TO_STRING(FLS));
	10..99:
		sFLS:=CONCAT(STR1:='FLS0' , STR2:= UINT_TO_STRING(FLS));
	100..999:
		sFLS:=CONCAT(STR1:='FLS' , STR2:= UINT_TO_STRING(FLS));
	ELSE
		;		
	END_CASE
	sString[8]:=CONCAT(STR1:=sFLS ,STR2:= ' ');
	
	sString[9]:=CONCAT(STR1:='FLR' , STR2:= UINT_TO_STRING(FLR));
	sString[10]:=CONCAT(STR1:=sString[9] ,STR2:= ' ');
	
	CASE FLK OF 
	0..9:
		sFLK:=CONCAT(STR1:='FLK00' , STR2:= UINT_TO_STRING(FLK));
	10..99:
		sFLK:=CONCAT(STR1:='FLK0' , STR2:= UINT_TO_STRING(FLK));
	100..999:
		sFLK:=CONCAT(STR1:='FLK' , STR2:= UINT_TO_STRING(FLK));
	ELSE
		;		
	END_CASE
	
	sString[12]:=CONCAT(STR1:=sFLK ,STR2:= ' ');
	

	CASE FLM OF 
	0..9:
		sFLM:=CONCAT(STR1:='FLM00' , STR2:= UINT_TO_STRING(FLM));
	10..99:
		sFLM:=CONCAT(STR1:='FLM0' , STR2:= UINT_TO_STRING(FLM));
	100..999:
		sFLM:=CONCAT(STR1:='FLM' , STR2:= UINT_TO_STRING(FLM));
	ELSE
		;		
	END_CASE
//	sString[14]:=CONCAT(STR1:=sFLM ,STR2:= ' ');
	sString[14]:=sFLM;

	sWString[0]:=CONCAT(STR1:=sString[0] ,STR2:= sString[2]);
	sWString[1]:=CONCAT(STR1:=sString[4] ,STR2:= sString[6]);
	sWString[2]:=CONCAT(STR1:=sString[8] ,STR2:= sString[10]);
	sWString[3]:=CONCAT(STR1:=sString[12] ,STR2:= sString[14]);
	
	sWString[6]:=CONCAT(STR1:=sWString[0] ,STR2:= sWString[1]);
	sWString[7]:=CONCAT(STR1:=sWString[2] ,STR2:= sWString[3]);
	sWString[8]:=CONCAT(STR1:=sWString[6] ,STR2:= sWString[7]);
	sWString[9]:=CONCAT(STR1:=sWString[8] ,STR2:= '03');
	sWString[10]:=CONCAT(STR1:=sWString[9] ,STR2:= ' ');
	
	Out:=sWString[8];

END_FUNCTION_BLOCK

// Device/Application/aSpecailBasic/String_TO_ASCII
FUNCTION_BLOCK String_TO_ASCII
VAR_INPUT
	InputString: STRING;          // 输入字符串
    MaxArraySize: INT := 255;    // 数组最大长度限制
END_VAR
VAR_OUTPUT
	 ASCIIArray: ARRAY[1..255] OF BYTE;  // 存储ASCII码的数组
     ArrayLength: INT;                 // 实际转换的字符数量
     Error: BOOL;                       // 错误标志
     ErrorMessage: STRING;              // 错误信息
END_VAR
VAR
	i: INT;  // 循环计数器
	sASCII_IN: INT;
	sSingleString:STRING;
END_VAR


    
    // 初始化输出
    Error := FALSE;
    ErrorMessage := '';
    ArrayLength := 0;
    
    // 检查输入字符串是否为空
    IF InputString = '' THEN
        Error := TRUE;
        ErrorMessage := '输入字符串为空';
        RETURN;
    END_IF;
    
    // 检查数组大小限制是否有效
    IF MaxArraySize < 1 OR MaxArraySize > 255 THEN
        Error := TRUE;
        ErrorMessage := '无效的数组大小限制';
        RETURN;
    END_IF;
    
    // 计算实际需要转换的字符数量（取字符串长度和最大数组大小的较小值）
    ArrayLength := MIN(LEN(InputString), MaxArraySize);
    
    // 转换每个字符为ASCII码并存储到数组
    FOR i := 1 TO ArrayLength DO
	   ASCIIArray[i] :=String2ASCII(sASCII_IN:=MID(InputString,1,i));
    END_FOR;

END_FUNCTION_BLOCK

// Device/Application/aSpecailBasic/String2ASCII
FUNCTION String2ASCII : BYTE

VAR_INPUT
	sASCII_IN:STRING;
END_VAR

VAR
	sIn_Single:STRING;
END_VAR

(*字符转换为16进制数字，BYTE数据类型*)

	sIn_Single:=LEFT(STR:=sASCII_IN , SIZE:=1 );//保证就一个字符
	
	IF    sIn_Single='A' THEN 	String2ASCII:=16#41;
	ELSIF sIn_Single='B' THEN  	String2ASCII:=16#42;
	ELSIF sIn_Single='C' THEN  	String2ASCII:=16#43;
	ELSIF sIn_Single='D' THEN	String2ASCII:=16#44;
	ELSIF sIn_Single='E' THEN	String2ASCII:=16#45;
	ELSIF sIn_Single='F' THEN	String2ASCII:=16#46;
	ELSIF sIn_Single='G' THEN	String2ASCII:=16#47;
	ELSIF sIn_Single='H' THEN	String2ASCII:=16#48;
	ELSIF sIn_Single='I' THEN	String2ASCII:=16#49;
	ELSIF sIn_Single='J' THEN	String2ASCII:=16#4A;
	ELSIF sIn_Single='K' THEN	String2ASCII:=16#4B;
	ELSIF sIn_Single='L' THEN	String2ASCII:=16#4C;
	ELSIF sIn_Single='M' THEN	String2ASCII:=16#4D;
	ELSIF sIn_Single='N' THEN	String2ASCII:=16#4E;
	ELSIF sIn_Single='O' THEN	String2ASCII:=16#4F;
	ELSIF sIn_Single='P' THEN	String2ASCII:=16#50;
	ELSIF sIn_Single='Q' THEN	String2ASCII:=16#51;
	ELSIF sIn_Single='R' THEN	String2ASCII:=16#52;
	ELSIF sIn_Single='S' THEN	String2ASCII:=16#53;
	ELSIF sIn_Single='T' THEN	String2ASCII:=16#54;
	ELSIF sIn_Single='U' THEN	String2ASCII:=16#55;
	ELSIF sIn_Single='V' THEN	String2ASCII:=16#56;
	ELSIF sIn_Single='W' THEN	String2ASCII:=16#57;
	ELSIF sIn_Single='X' THEN	String2ASCII:=16#58;
	ELSIF sIn_Single='Y' THEN	String2ASCII:=16#59;
	ELSIF sIn_Single='Z' THEN	String2ASCII:=16#5A;
	ELSIF sIn_Single='[' THEN	String2ASCII:=16#5B;
	ELSIF sIn_Single='\' THEN	String2ASCII:=16#5C;
	ELSIF sIn_Single=']' THEN	String2ASCII:=16#5D;
	ELSIF sIn_Single='^' THEN	String2ASCII:=16#5E;
	ELSIF sIn_Single='_' THEN	String2ASCII:=16#5F;
	ELSIF sIn_Single='`' THEN	String2ASCII:=16#60;
	
	ELSIF sIn_Single='a' THEN	String2ASCII:=16#61;	
	ELSIF sIn_Single='b' THEN  	String2ASCII:=16#62;
	ELSIF sIn_Single='c' THEN  	String2ASCII:=16#63;
	ELSIF sIn_Single='d' THEN	String2ASCII:=16#64;
	ELSIF sIn_Single='e' THEN	String2ASCII:=16#65;
	ELSIF sIn_Single='f' THEN	String2ASCII:=16#66;
	ELSIF sIn_Single='g' THEN	String2ASCII:=16#67;
	ELSIF sIn_Single='h' THEN	String2ASCII:=16#68;
	ELSIF sIn_Single='i' THEN	String2ASCII:=16#69;
	ELSIF sIn_Single='j' THEN	String2ASCII:=16#6A;
	ELSIF sIn_Single='k' THEN	String2ASCII:=16#6B;
	ELSIF sIn_Single='l' THEN	String2ASCII:=16#6C;
	ELSIF sIn_Single='m' THEN	String2ASCII:=16#6D;
	ELSIF sIn_Single='n' THEN	String2ASCII:=16#6E;
	ELSIF sIn_Single='o' THEN	String2ASCII:=16#6F;
	ELSIF sIn_Single='p' THEN	String2ASCII:=16#70;
	ELSIF sIn_Single='q' THEN	String2ASCII:=16#71;
	ELSIF sIn_Single='r' THEN	String2ASCII:=16#72;
	ELSIF sIn_Single='s' THEN	String2ASCII:=16#73;
	ELSIF sIn_Single='t' THEN	String2ASCII:=16#74;
	ELSIF sIn_Single='u' THEN	String2ASCII:=16#75;
	ELSIF sIn_Single='v' THEN	String2ASCII:=16#76;
	ELSIF sIn_Single='w' THEN	String2ASCII:=16#77;
	ELSIF sIn_Single='x' THEN	String2ASCII:=16#78;
	ELSIF sIn_Single='y' THEN	String2ASCII:=16#79;
	ELSIF sIn_Single='z' THEN	String2ASCII:=16#7A;
	ELSIF sIn_Single='{' THEN	String2ASCII:=16#7B;
	ELSIF sIn_Single='|' THEN	String2ASCII:=16#7C;
	ELSIF sIn_Single='}' THEN	String2ASCII:=16#7D;
	
	ELSIF sIn_Single='0' THEN  	String2ASCII:=16#30;
	ELSIF sIn_Single='1' THEN  	String2ASCII:=16#31;
	ELSIF sIn_Single='2' THEN	String2ASCII:=16#32;
	ELSIF sIn_Single='3' THEN	String2ASCII:=16#33;
	ELSIF sIn_Single='4' THEN	String2ASCII:=16#34;
	ELSIF sIn_Single='5' THEN	String2ASCII:=16#35;
	ELSIF sIn_Single='6' THEN	String2ASCII:=16#36;
	ELSIF sIn_Single='7' THEN	String2ASCII:=16#37;
	ELSIF sIn_Single='8' THEN	String2ASCII:=16#38;
	ELSIF sIn_Single='9' THEN	String2ASCII:=16#39;
	ELSIF sIn_Single=':' THEN	String2ASCII:=16#3A;
	ELSIF sIn_Single=';' THEN	String2ASCII:=16#3B;
	ELSIF sIn_Single='<' THEN	String2ASCII:=16#3C;
	ELSIF sIn_Single='=' THEN	String2ASCII:=16#3D;
	ELSIF sIn_Single='>' THEN	String2ASCII:=16#3E;
	ELSIF sIn_Single='?' THEN	String2ASCII:=16#3F;
	ELSIF sIn_Single='@' THEN	String2ASCII:=16#40;
		
	ELSIF sIn_Single=' ' THEN	String2ASCII:=16#20;	
	ELSIF sIn_Single='!' THEN	String2ASCII:=16#21;
	ELSIF sIn_Single='"' THEN	String2ASCII:=16#22;
	ELSIF sIn_Single='#' THEN	String2ASCII:=16#23;
//	ELSIF sIn_Single='$' THEN	String2ASCII:=16#24;
	ELSIF sIn_Single='%' THEN	String2ASCII:=16#25;
	ELSIF sIn_Single='&' THEN	String2ASCII:=16#26;
//	ELSIF sIn_Single=''' THEN	String2ASCII:=16#27;
	ELSIF sIn_Single='(' THEN	String2ASCII:=16#28;
	ELSIF sIn_Single=')' THEN	String2ASCII:=16#29;
	ELSIF sIn_Single='*' THEN	String2ASCII:=16#2A;
	ELSIF sIn_Single='+' THEN	String2ASCII:=16#2B;
	ELSIF sIn_Single=',' THEN	String2ASCII:=16#2C;
	ELSIF sIn_Single='-' THEN	String2ASCII:=16#2D;
	ELSIF sIn_Single='.' THEN	String2ASCII:=16#2E;
	ELSIF sIn_Single='/' THEN	String2ASCII:=16#2F;
	ELSE
		String2ASCII:=16#FF;	 //错误标志
	END_IF

END_FUNCTION

// Device/Application/aSpecailBasic/X_RayExpPara
FUNCTION_BLOCK X_RayExpPara
VAR_INPUT
	WS:UINT;  //工作站
	FO:UINT;//焦点
	ET:UINT;//曝光模式，MAS方式
	FI:UINT;//AEC选择
	FS:UINT;
	FN:UINT;//AEC DENSITY
	KV:UINT; //电压
	MA:UDINT;//电流
	MS:UDINT;//曝光时间
END_VAR
VAR_OUTPUT
	Out:STRING;
END_VAR
VAR
	sString :ARRAY [0..15] OF STRING;
	sWString :ARRAY [0..15] OF STRING;
	
	sKV,sMA,sMS:STRING;
END_VAR

(*Readme*)
(*曝光模式下大命令组合命令*)

	sString[0]:=CONCAT(STR1:='SA' , STR2:= ' ');
	
	sString[1]:=CONCAT(STR1:='WS' , STR2:= UINT_TO_STRING(WS));
	sString[2]:=CONCAT(STR1:=sString[1] ,STR2:= ' ');
	
	sString[3]:=CONCAT(STR1:='FO' , STR2:= UINT_TO_STRING(FO));
	sString[4]:=CONCAT(STR1:=sString[3] ,STR2:= ' ');
	
	sString[5]:=CONCAT(STR1:='ET' , STR2:= UINT_TO_STRING(ET));
	sString[6]:=CONCAT(STR1:=sString[5] ,STR2:= ' ');
	
	sString[7]:=CONCAT(STR1:='FI000',STR2:= ' ');
	
	sString[8]:=CONCAT(STR1:='FS001',STR2:= ' ');
	
	sString[9]:=CONCAT(STR1:='FN+0',STR2:= ' ');
	

	CASE KV OF 
	0..9:
		sKV:=CONCAT(STR1:='KV00' , STR2:= UINT_TO_STRING(LIMIT(40,KV,150)));
	10..99:
		sKV:=CONCAT(STR1:='KV0' , STR2:= UINT_TO_STRING(LIMIT(40,KV,150)));
	100..999:
		sKV:=CONCAT(STR1:='KV' , STR2:= UINT_TO_STRING(LIMIT(40,KV,150)));
	ELSE
		;		
	END_CASE
	sString[10]:=CONCAT(STR1:=sKV ,STR2:= ' ');
	

	CASE MA OF 
	0..9:
		sMA:=CONCAT(STR1:='MA0000' , STR2:= UDINT_TO_STRING(MA));
	10..99:
		sMA:=CONCAT(STR1:='MA000' , STR2:= UDINT_TO_STRING(MA));
	100..999:
		sMA:=CONCAT(STR1:='MA00' , STR2:= UDINT_TO_STRING(MA));
	1000..9999:
		sMA:=CONCAT(STR1:='MA0' , STR2:= UDINT_TO_STRING(MA));
	10000..99999:
		sMA:=CONCAT(STR1:='MA' , STR2:= UDINT_TO_STRING(MA));
	ELSE
		;		
	END_CASE
	sString[12]:=CONCAT(STR1:=sMA ,STR2:= ' ');

	CASE MS OF 
	0..9:
		sMS:=CONCAT(STR1:='MS0000' , STR2:= UDINT_TO_STRING(MS));
	10..99:
		sMS:=CONCAT(STR1:='MS000' , STR2:= UDINT_TO_STRING(MS));
	100..999:
		sMS:=CONCAT(STR1:='MS00' , STR2:= UDINT_TO_STRING(MS));
	1000..9999:
		sMS:=CONCAT(STR1:='MS0' , STR2:= UDINT_TO_STRING(MS));
	10000..99999:
		sMS:=CONCAT(STR1:='MS' , STR2:= UDINT_TO_STRING(MS));
	ELSE
		;		
	END_CASE
	sString[14]:=sMS;
//	sString[14]:=CONCAT(STR1:=sMS ,STR2:= ' ');

	(*组合*)
	sWString[0]:=CONCAT(STR1:=sString[0] ,STR2:= sString[2]);
	sWString[1]:=CONCAT(STR1:=sString[4] ,STR2:= sString[6]);
	sWString[2]:=CONCAT(STR1:=sString[7] ,STR2:= sString[8]);
	sWString[3]:=CONCAT(STR1:=sString[9] ,STR2:= sString[10]);
	sWString[4]:=CONCAT(STR1:=sString[12] ,STR2:= sString[14]);
	
	sWString[6]:=CONCAT(STR1:=sWString[0] ,STR2:= sWString[1]);
	sWString[7]:=CONCAT(STR1:=sWString[2] ,STR2:= sWString[3]);
	sWString[8]:=CONCAT(STR1:=sWString[7] ,STR2:= sWString[4]);
	
	
	sWString[9]:=CONCAT(STR1:=sWString[6] ,STR2:= sWString[8]);
//	sWString[10]:=CONCAT(STR1:=sWString[9] ,STR2:= sWString[8]);
	
	
	
	Out:=sWString[9];
//	Out:=sWString[10];

END_FUNCTION_BLOCK

// Device/Application/Communication/WorkStation_TCP
PROGRAM WorkStation_TCP
VAR
	count:BYTE;
	BOOTING:BOOL:=TRUE;
	TCP_Client_1: NBS.TCP_Client;
	TCP_Server_1: NBS.TCP_Server;
	TCP_Connection_1: NBS.TCP_Connection;
	TCP_Read_1: NBS.TCP_Read;
	TCP_Write_1:NBS.TCP_Write;
	IP:NBS.IP_ADDR;
	ServeruiPort:UINT:=8900;
	xTCP_Client_Enable:BOOL;
	hServer:CAA.HANDLE;
	hConn:CAA.HANDLE;
	
	abyWriteData:ARRAY[0..119] OF BYTE;
	abyReadData:ARRAY[0..119] OF BYTE;
	TON1,TON2:TON;BLINK1:Blink;
	TOF1:TOF;//延迟赋值socket 0
	
	RealByte1	:ARRAY[0..12] OF Real_TO_Byte_Convert;
	RealByte2	:ARRAY[0..12] OF Real_TO_Byte_Convert;
	
	bSetServerIP:BOOL;
	iServerIP1,iServerIP2,iServerIP3,iServerIP4:INT;
	TEMP_IP1,TEMP_IP2,TEMP_IP3,TEMP_IP4,TEMP_IP5:STRING;
	
	PLC_RECV_TEMP:PLC_RECV;//增加缓存
	
	R_TRIG_Trigger:R_TRIG;
	
	XZ_Error,QJ_Error:UDINT;
END_VAR

VAR_INPUT
	PLC_SEND1:PLC_SEND;
END_VAR

VAR_OUTPUT	
	PLC_RECV1:PLC_RECV;
	Socket:UDINT;
END_VAR

(*-------------------README----------------------*)
(*0.与上位机通讯并进行数据解析功能*)
(*1.PLC是客户机，IP：192.168.8.100：8899*)	//远程主机
(*2.工作站是服务器，IP：192.168.8.188：8900*)
	
(*0.心跳*)
	count:=count+1;
	
	IF BOOTING THEN  //有风险，可能无法写入数值了 iServerIP4<>0
		IP.sAddr:='192.168.10.20';
		BOOTING:=FALSE;
	END_IF
	
	IF hConn=0 THEN
		BLINK1(ENABLE:=TRUE , TIMELOW:=T#2S , TIMEHIGH:=T#4S , OUT=>xTCP_Client_Enable );
	ELSE
		BLINK1(ENABLE:=FALSE);
		xTCP_Client_Enable:=TRUE;
	END_IF
	
(*0.1 设置服务器IP及端口号*)
	IF bSetServerIP THEN
		TEMP_IP1:=Standard.CONCAT(INT_TO_STRING(iServerIP1),'.');
		TEMP_IP2:=Standard.CONCAT(INT_TO_STRING(iServerIP2),'.');
		TEMP_IP3:=Standard.CONCAT(INT_TO_STRING(iServerIP3),'.');
		TEMP_IP4:=Standard.CONCAT(TEMP_IP3,INT_TO_STRING(iServerIP4));
		TEMP_IP5:=Standard.CONCAT(TEMP_IP1,TEMP_IP2);
		IP.sAddr:=Standard.CONCAT(TEMP_IP5,TEMP_IP4);
		ServeruiPort:=ServeruiPort;
	END_IF
	
(*1.与服务器建立连接*)
	TCP_Connection_1(	
				xEnable:= xTCP_Client_Enable, 
				hServer:= hServer,
				xDone=> , 
				xBusy=> , 
				xError=> ,  
				eError=> , 
				xActive=> , 
				hConnection=> );
	
(*2.客户机设置*)
	TCP_Client_1(
				xEnable:= xTCP_Client_Enable , 
				xDone=> , 
				xBusy=> , 
				xError=> , 
				udiTimeOut:=500000 , 
				ipAddr:=IP , 	//客户端所连接的服务器IP地址
				uiPort:= ServeruiPort, //客户端所连接的服务器端口号
				eError=> , 
				xActive=> , 
				hConnection=>hConn );
				
(*3.读取数据*)
	TCP_Read_1(
				xEnable:=TON1.Q AND TCP_Client_1.xBusy , 
				xDone=> , 
				xBusy=> , 
				xError=> , 
				hConnection:= hConn, 
				szSize:= 120, 
				pData:=ADR(abyReadData) , 
				eError=> , 
				xReady=> , 
				szCount=> );
				
(*4.写入数据并发送*)
	R_TRIG_Trigger(CLK:=WorkStation_TCP.PLC_SEND1.m_nExpStates=2 AND GVL_State.iPLC_State=240 , Q=> );
	TCP_Write_1(
				xExecute:= (TON1.Q OR R_TRIG_Trigger.Q) AND TCP_Client_1.xBusy, 
				udiTimeOut:= 500000, 
				xDone=> , 
				xBusy=> , 
				xError=> , 
				hConnection:= hConn, 
				szSize:= 120, 
				pData:= ADR(abyWriteData), 
				eError=> );
				
(*5.设计发送和接收周期*)				
	TON1(IN:=NOT TON1.Q , PT:=T#200MS , Q=> , ET=> );
	
(*6.启动发送和接收数据*)
	APLC_RECV();
	APLC_SENG();

ACTION APLC_RECV:

(*----------------------PLC接收数据---------------------------*)//大端接收
(*1.//0为连接判断信息使用，1为发送设备的有具体意义是参数信息*)
	PLC_RECV_TEMP.m_nSocketType	:=BYTE_TO_UDINT(abyReadData[0])+ROL(BYTE_TO_UDINT(abyReadData[1]),8)+ROL(BYTE_TO_UDINT(abyReadData[2]),16)+ROL(BYTE_TO_UDINT(abyReadData[3]),24);
	
(*2.//扫描方式 0为不扫描， 1为定位像扫描； 2为CBCT扫描；3为DR扫描，4为快速扫描，5为旋转电机走到零位*)
	PLC_RECV_TEMP.m_nExpId		:=BYTE_TO_UDINT(abyReadData[4])+ROL(BYTE_TO_UDINT(abyReadData[5]),8)+ROL(BYTE_TO_UDINT(abyReadData[6]),16)+ROL(BYTE_TO_UDINT(abyReadData[7]),24);
	
(*3.//为曝光起始位置，在2D和多次曝光情况下，机架旋转到m_nAngleStart位置后再开始曝光，机架不动；CBCT状态下，机架旋转到m_nAngleStart位置后开始曝光，机架运动至m_nAngleEnd位置；最小值为0。*)
	RealByte2[0].wByte[0]:=abyReadData[8];
	RealByte2[0].wByte[1]:=abyReadData[9];
	RealByte2[0].wByte[2]:=abyReadData[10];
	RealByte2[0].wByte[3]:=abyReadData[11];
	PLC_RECV_TEMP.m_nAngleStart	:=RealByte2[0].rData;

(*4.//为曝光的终止位置，在2D和多次曝光情况下不使用；在CBCT状态下，机架的运动终止位置；最小值为0，最大值为360。*)
	RealByte2[1].wByte[0]:=abyReadData[12];
	RealByte2[1].wByte[1]:=abyReadData[13];
	RealByte2[1].wByte[2]:=abyReadData[14];
	RealByte2[1].wByte[3]:=abyReadData[15];
	PLC_RECV_TEMP.m_nAngleEnd	:=RealByte2[1].rData;

(*5.//为旋转的起始位置（考虑加速过程）*)
	RealByte2[2].wByte[0]:=abyReadData[16];
	RealByte2[2].wByte[1]:=abyReadData[17];
	RealByte2[2].wByte[2]:=abyReadData[18];
	RealByte2[2].wByte[3]:=abyReadData[19];
	PLC_RECV_TEMP.m_nRotateBegin	:=RealByte2[2].rData;
	
(*6.//为旋转的终止位置（考虑减速过程）*)
	RealByte2[3].wByte[0]:=abyReadData[20];
	RealByte2[3].wByte[1]:=abyReadData[21];
	RealByte2[3].wByte[2]:=abyReadData[22];
	RealByte2[3].wByte[3]:=abyReadData[23];
	PLC_RECV_TEMP.m_nRotateEnd	:=RealByte2[3].rData;

(*7.//设置的管电压值，单位为kv，正整数；*)
	PLC_RECV_TEMP.m_nKv	:=BYTE_TO_UDINT(abyReadData[24])+ROL(BYTE_TO_UDINT(abyReadData[25]),8)+ROL(BYTE_TO_UDINT(abyReadData[26]),16)+ROL(BYTE_TO_UDINT(abyReadData[27]),24);

(*8.//设置的管电流值，单位为mA，正整数；*)
	RealByte2[5].wByte[0]:=abyReadData[28];
	RealByte2[5].wByte[1]:=abyReadData[29];
	RealByte2[5].wByte[2]:=abyReadData[30];
	RealByte2[5].wByte[3]:=abyReadData[31];
	PLC_RECV_TEMP.m_nMA	:=RealByte2[5].rData;

(*9.//设置一次曝光的时间，单位为MS（毫秒）；*)
	RealByte2[6].wByte[0]:=abyReadData[32];
	RealByte2[6].wByte[1]:=abyReadData[33];
	RealByte2[6].wByte[2]:=abyReadData[34];
	RealByte2[6].wByte[3]:=abyReadData[35];
	PLC_RECV_TEMP.m_nMS	:=RealByte2[6].rData;

(*10.//焦点大小设置，枚举值，0为大焦点， 1小焦点；*)
	PLC_RECV_TEMP.m_nFocus:=BYTE_TO_UDINT(abyReadData[36]);
	
(*11.//总帧数，正整数；*)
	PLC_RECV_TEMP.m_nAcquireFrame 	:=BYTE_TO_UDINT(abyReadData[40])+ROL(BYTE_TO_UDINT(abyReadData[41]),8)+ROL(BYTE_TO_UDINT(abyReadData[42]),16)+ROL(BYTE_TO_UDINT(abyReadData[43]),24);	
	
(*12.//每圈获得的帧数，正整数，帧/圈；*)	
	PLC_RECV_TEMP.m_nFramePerCirCle	:=BYTE_TO_UDINT(abyReadData[44])+ROL(BYTE_TO_UDINT(abyReadData[45]),8)+ROL(BYTE_TO_UDINT(abyReadData[46]),16)+ROL(BYTE_TO_UDINT(abyReadData[47]),24);	
	
(*13.扫描方向，0为不移动，1为进床方向，2为出床方向；*)	
	PLC_RECV_TEMP.m_nMoveToward		:=BYTE_TO_UDINT(abyReadData[48])+ROL(BYTE_TO_UDINT(abyReadData[49]),8)+ROL(BYTE_TO_UDINT(abyReadData[50]),16)+ROL(BYTE_TO_UDINT(abyReadData[51]),24);
	
(*14.//7灯是否点亮；*)
	PLC_RECV_TEMP.m_nServenLamp 	:=BYTE_TO_UDINT(abyReadData[52])+ROL(BYTE_TO_UDINT(abyReadData[53]),8)+ROL(BYTE_TO_UDINT(abyReadData[54]),16)+ROL(BYTE_TO_UDINT(abyReadData[55]),24);
	
	
(*15//步进长度，轴扫时使用，单位为mm（毫米）；*)
	RealByte2[4].wByte[0]:=abyReadData[56];
	RealByte2[4].wByte[1]:=abyReadData[57];
	RealByte2[4].wByte[2]:=abyReadData[58];
	RealByte2[4].wByte[3]:=abyReadData[59];
	PLC_RECV_TEMP.m_nMoveStep:=RealByte2[4].rData;
	
(*16//螺距长度，螺旋扫时使用，单位为mm（毫米）；*)
	RealByte2[7].wByte[0]:=abyReadData[60];
	RealByte2[7].wByte[1]:=abyReadData[61];
	RealByte2[7].wByte[2]:=abyReadData[62];
	RealByte2[7].wByte[3]:=abyReadData[63];
	PLC_RECV_TEMP.m_nPitchValue	:=RealByte2[7].rData;
	
(*17//旋转总圈数，由起始角度和终止角度计算获得，正整数。*)
	PLC_RECV_TEMP.m_nCircleCount  	:=BYTE_TO_UDINT(abyReadData[64])+ROL(BYTE_TO_UDINT(abyReadData[65]),8)+ROL(BYTE_TO_UDINT(abyReadData[66]),16)+ROL(BYTE_TO_UDINT(abyReadData[67]),24);
	
(*18//控制状态 0为正常 1为中止扫描， 2为退出扫描，默认为0*)
	PLC_RECV_TEMP.m_nControlState  	:=BYTE_TO_UDINT(abyReadData[68])+ROL(BYTE_TO_UDINT(abyReadData[69]),8)+ROL(BYTE_TO_UDINT(abyReadData[70]),16)+ROL(BYTE_TO_UDINT(abyReadData[71]),24);

(*19//扫描上界，以动物趴卧头朝里的方向为基准，从脚至头方向为正方向。单位为毫米，精度为0.01；*)
	RealByte2[8].wByte[0]:=abyReadData[72];
	RealByte2[8].wByte[1]:=abyReadData[73];
	RealByte2[8].wByte[2]:=abyReadData[74];
	RealByte2[8].wByte[3]:=abyReadData[75];
	PLC_RECV_TEMP.m_fScanTop	:=RealByte2[8].rData;//零点偏移
	
(*20///扫描下界，以动物趴卧头朝里的方向为基准，从脚至头方向为正方向。单位为毫米，精度为0.01；*)
	RealByte2[9].wByte[0]:=abyReadData[76];
	RealByte2[9].wByte[1]:=abyReadData[77];
	RealByte2[9].wByte[2]:=abyReadData[78];
	RealByte2[9].wByte[3]:=abyReadData[79];
	PLC_RECV_TEMP.m_fScanBottom	:=RealByte2[9].rData;//零点偏移;
	
(*21////一圈多少秒*)
	RealByte2[11].wByte[0]:=abyReadData[80];
	RealByte2[11].wByte[1]:=abyReadData[81];
	RealByte2[11].wByte[2]:=abyReadData[82];
	RealByte2[11].wByte[3]:=abyReadData[83];
	PLC_RECV_TEMP.m_fSecondPerCicle	:=RealByte2[11].rData;//一圈多少秒*)
//	PLC_RECV_TEMP.m_fSecondPerCicle  :=BYTE_TO_UDINT(abyReadData[80])+ROL(BYTE_TO_UDINT(abyReadData[81]),8)+ROL(BYTE_TO_UDINT(abyReadData[82]),16)+ROL(BYTE_TO_UDINT(abyReadData[83]),24);
		
(*22//采样率，有3个选项：2400帧/圈；1200帧/圈；600帧/圈*)
	PLC_RECV_TEMP.m_nSamplingRate  	:=BYTE_TO_UDINT(abyReadData[84])+ROL(BYTE_TO_UDINT(abyReadData[85]),8)+ROL(BYTE_TO_UDINT(abyReadData[86]),16)+ROL(BYTE_TO_UDINT(abyReadData[87]),24);	

(*23//是否亮灯1为亮5灯，0 为不亮5灯*)
	PLC_RECV_TEMP.m_nPrepareState  	:=BYTE_TO_UDINT(abyReadData[88])+ROL(BYTE_TO_UDINT(abyReadData[89]),8)+ROL(BYTE_TO_UDINT(abyReadData[90]),16)+ROL(BYTE_TO_UDINT(abyReadData[91]),24);

(*24////扫描模式 0为手动扫描，1为自动扫描，2为子床位扫描*)
	PLC_RECV_TEMP.m_nScanMoveType  	:=BYTE_TO_UDINT(abyReadData[92])+ROL(BYTE_TO_UDINT(abyReadData[93]),8)+ROL(BYTE_TO_UDINT(abyReadData[94]),16)+ROL(BYTE_TO_UDINT(abyReadData[95]),24);

(*25//当前第几圈*)
	PLC_RECV_TEMP.m_nCircleIndex  	:=BYTE_TO_UDINT(abyReadData[96])+ROL(BYTE_TO_UDINT(abyReadData[97]),8)+ROL(BYTE_TO_UDINT(abyReadData[98]),16)+ROL(BYTE_TO_UDINT(abyReadData[99]),24);
		
(*26//灯丝电压值*)
	RealByte2[10].wByte[0]:=abyReadData[100];
	RealByte2[10].wByte[1]:=abyReadData[101];
	RealByte2[10].wByte[2]:=abyReadData[102];
	RealByte2[10].wByte[3]:=abyReadData[103];
	PLC_RECV_TEMP.m_nPLCMaCoeff	:=RealByte2[10].rData;	

(*27//CBCT扫描最后一次标志位*)
	PLC_RECV_TEMP.m_nLastMsg  	:=BYTE_TO_UDINT(abyReadData[104])+ROL(BYTE_TO_UDINT(abyReadData[105]),8)+ROL(BYTE_TO_UDINT(abyReadData[106]),16)+ROL(BYTE_TO_UDINT(abyReadData[107]),24);
	
(*28//预留*)
	PLC_RECV_TEMP.m_nDelayTime	:=BYTE_TO_UDINT(abyReadData[108])+ROL(BYTE_TO_UDINT(abyReadData[109]),8)+ROL(BYTE_TO_UDINT(abyReadData[110]),16)+ROL(BYTE_TO_UDINT(abyReadData[111]),24);//预留//预留一共30个数据
	PLC_RECV_TEMP.yuliu_2		:=BYTE_TO_UDINT(abyReadData[112])+ROL(BYTE_TO_UDINT(abyReadData[113]),8)+ROL(BYTE_TO_UDINT(abyReadData[114]),16)+ROL(BYTE_TO_UDINT(abyReadData[115]),24);//预留//预留一共30个数据
	PLC_RECV_TEMP.yuliu_3		:=BYTE_TO_UDINT(abyReadData[116])+ROL(BYTE_TO_UDINT(abyReadData[117]),8)+ROL(BYTE_TO_UDINT(abyReadData[118]),16)+ROL(BYTE_TO_UDINT(abyReadData[119]),24);//预留//预留一共30个数据


(*---------------------------------------缓存处理------------------------------*)
Socket:=PLC_RECV_TEMP.m_nSocketType;
IF PLC_RECV_TEMP.m_nSocketType=1 THEN
    PLC_RECV1:=PLC_RECV_TEMP;
	TOF1(IN:=FALSE);
ELSE
	TOF1(IN:=TRUE , PT:=T#150MS, Q=> , ET=> );
	IF TOF1.Q THEN
		PLC_RECV1.m_nSocketType		:=	PLC_RECV_TEMP.m_nSocketType	;
	ELSE
		PLC_RECV1.m_nSocketType		:=	PLC_RECV1.m_nSocketType	;
	END_IF
	
	PLC_RECV1.m_nExpId 			:=  PLC_RECV1.m_nExpId 			;      
	PLC_RECV1.m_nAngleStart 	:=	PLC_RECV1.m_nAngleStart 	;   
	PLC_RECV1.m_nAngleEnd  		:=	PLC_RECV1.m_nAngleEnd  		;   
	PLC_RECV1.m_nRotateBegin  	:=  PLC_RECV1.m_nRotateBegin  	; 
	PLC_RECV1.m_nRotateEnd  	:=	PLC_RECV1.m_nRotateEnd  	;   
	PLC_RECV1.m_nKv  			:=	PLC_RECV1.m_nKv  			;       
	PLC_RECV1.m_nMA  			:=	PLC_RECV1.m_nMA  			;        
	PLC_RECV1.m_nMS 			:=	PLC_RECV1.m_nMS 			;        
	PLC_RECV1.m_nFocus 			:=  PLC_RECV1.m_nFocus 			;     
	PLC_RECV1.m_nAcquireFrame 	:=  PLC_RECV1.m_nAcquireFrame 	;
	PLC_RECV1.m_nFramePerCirCle	:=  PLC_RECV1.m_nFramePerCirCle	;
	PLC_RECV1.m_nMoveToward  	:=	PLC_RECV1.m_nMoveToward  	 ;
	PLC_RECV1.m_nServenLamp  	:=  PLC_RECV1.m_nServenLamp  	 ;
	PLC_RECV1.m_nMoveStep  		:=  PLC_RECV1.m_nMoveStep  		 ;  
	PLC_RECV1.m_nPitchValue   	:=  PLC_RECV1.m_nPitchValue   	 ;
	PLC_RECV1.m_nCircleCount  	:=  PLC_RECV1.m_nCircleCount  	 ;
	PLC_RECV1.m_nControlState 	:=  PLC_RECV1.m_nControlState 	 ;
	PLC_RECV1.m_fScanTop 		:=	PLC_RECV1.m_fScanTop 		 ;    
	PLC_RECV1.m_fScanBottom 	:=	PLC_RECV1.m_fScanBottom 	 ;  
	PLC_RECV1.m_fSecondPerCicle	:=  PLC_RECV1.m_fSecondPerCicle	;
	PLC_RECV1.m_nSamplingRate  	:=  PLC_RECV1.m_nSamplingRate  	;
	PLC_RECV1.m_nPrepareState 	:=  PLC_RECV1.m_nPrepareState 	 ;
	PLC_RECV1.m_nScanMoveType	:=	PLC_RECV1.m_nScanMoveType	;  
	PLC_RECV1.m_nCircleIndex 	:=	PLC_RECV1.m_nCircleIndex 	;  
	PLC_RECV1.m_nPLCMaCoeff 	:=	PLC_RECV1.m_nPLCMaCoeff 	 ;  
	PLC_RECV1.m_nLastMsg  		:=  PLC_RECV1.m_nLastMsg  		;    
	PLC_RECV1.m_nDelayTime 		:=  PLC_RECV1.m_nDelayTime 		;       
	PLC_RECV1.yuliu_2			:=	PLC_RECV1.yuliu_2			 ;       
	PLC_RECV1.yuliu_3 			:=  PLC_RECV1.yuliu_3 			 ;      	
END_IF
END_ACTION

ACTION APLC_SENG:

(*---------------------------------PLC发送数据------------------------------------*)//大端发送机制
(*第一部分，发送数据赋值,待补充*)
	IF PLC_RECV1.m_nSocketType=1 THEN
    	PLC_SEND1.m_nSocketType	  := 1;//心跳指令，默认为3，留待判断连接状态。
	ELSE
    	PLC_SEND1.m_nSocketType	  := 3;//心跳指令，默认为3，留待判断连接状态。
	END_IF                                                                            
	PLC_SEND1.m_nCurrentAngle	:= LREAL_TO_REAL(Axis_XZ.XZ_AxisState.rActPosition);//为设备当前的旋转角度，单位为角度制下的单位，为度。数精度为1度；                                                             
	PLC_SEND1.m_nBedHeight		:= Entity_IO.rRealPos; //为床高，单位为毫米，数据范围为0 - 2000mm；                                                                 
	PLC_SEND1.m_nBedMovePos		:= LREAL_TO_REAL(Axis_QJ.QJ_AxisState.rActPosition);//为床移动距离，以床与探测板的垂直面交线为起点，单位为毫米，数据范围为0 - 3000mm；//增加了偏移                                                 
//	PLC_SEND1.m_nExpStates		:= 22;//为曝光状态，枚举值，0:idle（空闲） 1:prep（训机） 2: ready（训机结束，准备完成，可以出束） 3: XrayOn（出射线） 4:XrayOff（关射线） 5 error；
	PLC_SEND1.m_nExpCount		:= PLC_PRG.iActNumPulse;//为曝光的次数，对应曝光的图像张数；                                                                              
//	PLC_SEND1.m_nFocus			:= XRAY_RS485.Feedback_nFocus;//焦点大小，0为大焦点 1为小焦点， 焦点具体对应的值由plc设置；        //修改为按键提示                                                      
	PLC_SEND1.m_nMHuValue		:= DT_Xray.Feedback_nMHuValue;//热容量，单位MHu ，实际热容量*100得到，实际热容量为小数；                                                               
//	PLC_SEND1.m_nDirectionState	:= 22;//当前旋转状态，默认值-1， 0为正转，1为反转，停止为-1                                                                  
//	PLC_SEND1.m_nMoveState		:= 22;//起始、终止状态， 默认值-1， 0为当前扫描方案（与常规意义不同，注意区别）处于准备好状态，可以准备扫描；1为当前扫描方案结束，运动过程中值为-1                      
	PLC_SEND1.m_nError			:= DT_Xray.iAlarmNum;//错误码使用，由王（风杰）工具体阐述内容                                                                            
	PLC_SEND1.m_fSpeed			:= LREAL_TO_REAL(Axis_XZ.XZ_AxisState.rActVelocity);//为设备的旋转速度，单位为度/秒，精度0.01度/秒；                                                                     
	PLC_SEND1.m_fKv				:= DT_Xray.Feedback_Kv;//管电压，单位为kv（千伏），精度0.01；                                                                          
	PLC_SEND1.m_fMA				:= DT_Xray.Feedback_mA;//管电流，单位为mA（毫安），精度0.01；                                                                          
	PLC_SEND1.m_fMs				:= DT_Xray.Feedback_ms;//曝光时间，单位为ms（毫秒），精度0.01；                                                                         
	PLC_SEND1.m_nSamplingRate	:= PLC_RECV1.m_nFramePerCirCle;//采样率，有3个选项：2400帧/圈；1200帧/圈；600帧/圈                                                               
//	PLC_SEND1.m_nScanProType	:= 22;//执行扫描方案的类型，0为自动扫描，1为手动扫描，2为无设置意义的值，默认值为2                                                        
	PLC_SEND1.PLC_State			:= GVL_State.iPLC_State;//PLC状态机状态                                                                                             
	PLC_SEND1.XRAY_State		:= GVL_State.iXray_State;//射线源状态                                                                                     
	PLC_SEND1.AxisErrorID		:= QJ_Error+XZ_Error*65536; //电机错误报警位,各占16位 
    PLC_SEND1.m_nFocusX			:= DT_Xray.Feedback_nFocus;//反馈jiao'dian

(**处理电机Errstop状态下没有故障吗的情况*)	
	IF Axis_XZ.XZ_AxisState.bAxisErr THEN
		XZ_Error:= Axis_XZ.XZ_AxisState.ErrorID ;
	ELSE
		IF  Axis_XZ.XZ_AxisState.bErrStop THEN
			XZ_Error:= 444 ; 
		ELSE
			XZ_Error:=0;
		END_IF
	END_IF
	
	IF Axis_QJ.QJ_AxisState.bAxisErr THEN
		XZ_Error:= Axis_QJ.QJ_AxisState.ErrorID ;
	ELSE
		IF  Axis_QJ.QJ_AxisState.bErrStop THEN
			QJ_Error:= 444 ; 
		ELSE
			QJ_Error:=0;
		END_IF
	END_IF
	                               
